C07311=1146.212,197.373,-62.411,-178.136,7.345,148.840
C07312=1146.216,197.124,-62.387,-178.138,7.343,148.841
C07313=1146.221,196.875,-62.364,-178.141,7.340,148.841
C07314=1146.225,196.626,-62.339,-178.144,7.338,148.841
C07315=1146.229,196.378,-62.315,-178.147,7.336,148.841
C07316=1146.234,196.129,-62.292,-178.149,7.334,148.842
C07317=1146.239,195.880,-62.267,-178.152,7.331,148.842
C07318=1146.244,195.631,-62.244,-178.155,7.328,148.842
C07319=1146.248,195.382,-62.220,-178.157,7.326,148.842
C07320=1146.253,195.133,-62.196,-178.161,7.324,148.843
C07321=1146.257,194.885,-62.172,-178.163,7.322,148.843
C07322=1146.261,194.635,-62.149,-178.166,7.319,148.843
C07323=1146.266,194.387,-62.124,-178.168,7.317,148.843
C07324=1146.271,194.137,-62.100,-178.172,7.314,148.844
C07325=1146.275,193.889,-62.076,-178.175,7.312,148.844
C07326=1146.280,193.640,-62.053,-178.177,7.310,148.844
C07327=1146.285,193.392,-62.029,-178.180,7.307,148.844
C07328=1146.289,193.143,-62.006,-178.183,7.305,148.845
C07329=1146.294,192.894,-61.982,-178.186,7.303,148.845
C07330=1146.298,192.645,-61.958,-178.188,7.300,148.845
C07331=1146.303,192.397,-61.934,-178.192,7.298,148.845
C07332=1146.307,192.148,-61.911,-178.194,7.296,148.845
C07333=1146.312,191.899,-61.887,-178.197,7.293,148.846
C07334=1146.317,191.650,-61.863,-178.199,7.291,148.846
C07335=1146.321,191.401,-61.840,-178.203,7.289,148.846
C07336=1146.326,191.152,-61.817,-178.205,7.287,148.846
C07337=1146.330,190.904,-61.793,-178.208,7.284,148.847
C07338=1146.335,190.655,-61.769,-178.211,7.281,148.847
C07339=1146.340,190.406,-61.746,-178.213,7.279,148.847
C07340=1146.344,190.157,-61.722,-178.216,7.276,148.847
C07341=1146.349,189.908,-61.698,-178.219,7.275,148.848
C07342=1146.354,189.659,-61.675,-178.222,7.272,148.848
C07343=1146.358,189.410,-61.652,-178.224,7.270,148.848
C07344=1146.363,189.162,-61.628,-178.228,7.267,148.848
C07345=1146.367,188.913,-61.604,-178.230,7.265,148.849
C07346=1146.372,188.664,-61.581,-178.233,7.263,148.849
C07347=1146.377,188.415,-61.558,-178.235,7.261,148.849
C07348=1146.381,188.166,-61.533,-178.239,7.258,148.849
C07349=1146.386,187.917,-61.510,-178.241,7.256,148.850
C07350=1146.391,187.668,-61.487,-178.244,7.254,148.850
C07351=1146.395,187.419,-61.463,-178.247,7.252,148.850
C07352=1146.399,187.170,-61.441,-178.250,7.249,148.850
C07353=1146.404,186.921,-61.417,-178.252,7.247,148.851
C07354=1146.409,186.672,-61.394,-178.255,7.244,148.851
C07355=1146.413,186.424,-61.370,-178.258,7.243,148.851
C07356=1146.418,186.175,-61.346,-178.261,7.240,148.851
C07357=1146.422,185.926,-61.323,-178.263,7.238,148.852
C07358=1146.426,185.677,-61.300,-178.267,7.235,148.852
C07359=1146.431,185.428,-61.277,-178.269,7.233,148.852
C07360=1146.436,185.180,-61.254,-178.272,7.231,148.853
C07361=1146.441,184.931,-61.231,-178.274,7.229,148.853
C07362=1146.446,184.682,-61.207,-178.278,7.226,148.853
C07363=1146.450,184.433,-61.184,-178.280,7.224,148.853
C07364=1146.454,184.184,-61.161,-178.283,7.221,148.853
C07365=1146.460,183.914,-61.136,-178.286,7.220,148.854
C07366=1146.465,183.644,-61.111,-178.289,7.217,148.854
C07367=1146.469,183.376,-61.086,-178.292,7.214,148.854
C07368=1146.475,183.106,-61.061,-178.295,7.212,148.855
C07369=1146.479,182.857,-61.037,-178.298,7.210,148.855
C07370=1146.484,182.608,-61.014,-178.301,7.207,148.855
C07371=1146.488,182.359,-60.991,-178.303,7.205,148.856
C07372=1146.493,182.110,-60.968,-178.307,7.203,148.856
C07373=1146.498,181.860,-60.945,-178.309,7.201,148.856
C07374=1146.502,181.612,-60.923,-178.312,7.198,148.856
C07375=1146.507,181.363,-60.900,-178.315,7.196,148.857
C07376=1146.512,181.114,-60.876,-178.317,7.194,148.857
C07377=1146.516,180.866,-60.853,-178.320,7.192,148.857
C07378=1146.520,180.617,-60.830,-178.323,7.190,148.857
C07379=1146.525,180.367,-60.807,-178.326,7.187,148.858
C07380=1146.530,180.119,-60.785,-178.329,7.185,148.858
C07381=1146.535,179.870,-60.762,-178.331,7.182,148.858
C07382=1146.539,179.621,-60.738,-178.334,7.181,148.859
C07383=1146.543,179.372,-60.716,-178.337,7.178,148.859
C07384=1146.548,179.122,-60.693,-178.340,7.176,148.859
C07385=1146.553,178.874,-60.671,-178.342,7.174,148.859
C07386=1146.558,178.625,-60.647,-178.346,7.172,148.860
C07387=1146.562,178.376,-60.624,-178.348,7.170,148.860
C07388=1146.566,178.127,-60.602,-178.351,7.167,148.860
C07389=1146.572,177.879,-60.579,-178.354,7.165,148.861
C07390=1146.576,177.630,-60.556,-178.357,7.163,148.861
C07391=1146.581,177.380,-60.533,-178.359,7.161,148.861
C07392=1146.585,177.132,-60.511,-178.362,7.159,148.861
C07393=1146.590,176.883,-60.488,-178.365,7.156,148.862
C07394=1146.594,176.634,-60.466,-178.368,7.154,148.862
C07395=1146.599,176.385,-60.442,-178.371,7.152,148.862
C07396=1146.603,176.135,-60.420,-178.373,7.150,148.862
C07397=1146.609,175.887,-60.397,-178.376,7.147,148.863
C07398=1146.613,175.638,-60.374,-178.379,7.146,148.863
C07399=1146.618,175.389,-60.352,-178.381,7.143,148.863
C07400=1146.622,175.141,-60.329,-178.385,7.141,148.864
C07401=1146.627,174.891,-60.307,-178.387,7.139,148.864
C07402=1146.631,174.642,-60.284,-178.390,7.136,148.864
C07403=1146.637,174.393,-60.262,-178.393,7.135,148.864
C07404=1146.641,174.145,-60.239,-178.395,7.133,148.865
C07405=1146.646,173.895,-60.216,-178.398,7.130,148.865
C07406=1146.650,173.647,-60.194,-178.401,7.128,148.865
C07407=1146.655,173.397,-60.171,-178.404,7.126,148.866
C07408=1146.659,173.149,-60.148,-178.406,7.124,148.866
C07409=1146.664,172.900,-60.127,-178.409,7.122,148.866
C07410=1146.669,172.651,-60.103,-178.412,7.119,148.867
C07411=1146.673,172.402,-60.081,-178.415,7.118,148.867
C07412=1146.679,172.153,-60.059,-178.418,7.115,148.867
C07413=1146.683,171.904,-60.036,-178.421,7.113,148.867
C07414=1146.687,171.655,-60.014,-178.423,7.111,148.868
C07415=1146.692,171.406,-59.991,-178.426,7.108,148.868
C07416=1146.696,171.157,-59.969,-178.429,7.107,148.868
C07417=1146.701,170.908,-59.948,-178.432,7.105,148.869
C07418=1146.706,170.659,-59.924,-178.435,7.102,148.869
C07419=1146.710,170.410,-59.902,-178.437,7.100,148.869
C07420=1146.715,170.161,-59.881,-178.440,7.098,148.870
C07421=1146.720,169.912,-59.857,-178.443,7.096,148.870
C07422=1146.725,169.664,-59.835,-178.445,7.094,148.870
C07423=1146.729,169.414,-59.813,-178.449,7.091,148.870
C07424=1146.735,169.165,-59.791,-178.451,7.090,148.871
C07425=1146.739,168.917,-59.768,-178.454,7.088,148.871
C07426=1146.743,168.667,-59.746,-178.457,7.085,148.871
C07427=1146.748,168.419,-59.725,-178.460,7.083,148.872
C07428=1146.753,168.169,-59.702,-178.462,7.081,148.872
C07429=1146.757,167.921,-59.680,-178.466,7.079,148.872
C07430=1146.761,167.672,-59.658,-178.468,7.077,148.872
C07431=1146.766,167.423,-59.636,-178.471,7.074,148.873
C07432=1146.771,167.173,-59.613,-178.474,7.073,148.873
C07433=1146.776,166.925,-59.592,-178.476,7.071,148.874
C07434=1146.781,166.675,-59.569,-178.479,7.068,148.874
C07435=1146.785,166.427,-59.548,-178.482,7.066,148.874
C07436=1146.790,166.178,-59.524,-178.485,7.065,148.874
C07437=1146.795,165.929,-59.503,-178.488,7.062,148.875
C07438=1146.799,165.680,-59.481,-178.490,7.060,148.875
C07439=1146.804,165.431,-59.459,-178.493,7.058,148.875
C07440=1146.808,165.182,-59.437,-178.496,7.056,148.876
C07441=1146.813,164.933,-59.415,-178.499,7.054,148.876
C07442=1146.817,164.684,-59.393,-178.501,7.052,148.876
C07443=1146.823,164.435,-59.371,-178.504,7.049,148.877
C07444=1146.827,164.185,-59.349,-178.507,7.048,148.877
C07445=1146.832,163.937,-59.327,-178.510,7.046,148.877
C07446=1146.837,163.687,-59.305,-178.513,7.043,148.878
C07447=1146.841,163.439,-59.284,-178.515,7.041,148.878
C07448=1146.846,163.189,-59.261,-178.518,7.039,148.878
C07449=1146.851,162.941,-59.240,-178.521,7.038,148.879
C07450=1146.855,162.692,-59.218,-178.524,7.035,148.879
C07451=1146.860,162.443,-59.196,-178.526,7.033,148.879
C07452=1146.865,162.194,-59.174,-178.529,7.031,148.879
C07453=1146.869,161.945,-59.152,-178.532,7.029,148.880
C07454=1146.874,161.696,-59.131,-178.535,7.027,148.880
C07455=1146.879,161.447,-59.108,-178.538,7.025,148.881
C07456=1146.884,161.198,-59.086,-178.540,7.023,148.881
C07457=1146.889,160.949,-59.065,-178.543,7.021,148.881
C07458=1146.893,160.699,-59.043,-178.546,7.019,148.881
C07459=1146.898,160.451,-59.022,-178.549,7.017,148.882
C07460=1146.902,160.201,-59.000,-178.552,7.015,148.882
C07461=1146.907,159.953,-58.978,-178.554,7.013,148.882
C07462=1146.912,159.704,-58.956,-178.557,7.011,148.883
C07463=1146.916,159.454,-58.935,-178.560,7.008,148.883
C07464=1146.921,159.206,-58.914,-178.563,7.007,148.883
C07465=1146.925,158.957,-58.892,-178.565,7.005,148.884
C07466=1146.930,158.708,-58.870,-178.569,7.003,148.884
C07467=1146.935,158.459,-58.848,-178.571,7.000,148.884
C07468=1146.939,158.209,-58.827,-178.574,6.999,148.885
C07469=1146.944,157.940,-58.803,-178.577,6.996,148.885
C07470=1146.950,157.672,-58.781,-178.580,6.994,148.886
C07471=1146.955,157.403,-58.757,-178.583,6.992,148.886
C07472=1146.960,157.134,-58.734,-178.586,6.990,148.886
C07473=1146.964,156.884,-58.712,-178.588,6.988,148.887
C07474=1146.969,156.636,-58.691,-178.592,6.986,148.887
C07475=1146.974,156.387,-58.669,-178.594,6.984,148.887
C07476=1146.978,156.137,-58.648,-178.597,6.982,148.888
C07477=1146.983,155.889,-58.626,-178.600,6.980,148.888
C07478=1146.989,155.639,-58.605,-178.603,6.978,148.888
C07479=1146.993,155.391,-58.584,-178.605,6.976,148.889
C07480=1146.997,155.142,-58.562,-178.608,6.974,148.889
C07481=1147.002,154.892,-58.541,-178.611,6.972,148.889
C07482=1147.007,154.644,-58.519,-178.614,6.970,148.890
C07483=1147.012,154.394,-58.498,-178.616,6.968,148.890
C07484=1147.016,154.145,-58.476,-178.619,6.966,148.890
C07485=1147.021,153.896,-58.456,-178.622,6.964,148.891
C07486=1147.026,153.647,-58.434,-178.625,6.962,148.891
C07487=1147.030,153.398,-58.413,-178.628,6.960,148.891
C07488=1147.035,153.149,-58.391,-178.630,6.959,148.892
C07489=1147.040,152.900,-58.371,-178.633,6.957,148.892
C07490=1147.044,152.651,-58.349,-178.636,6.954,148.892
C07491=1147.050,152.402,-58.328,-178.639,6.952,148.893
C07492=1147.054,152.153,-58.306,-178.641,6.951,148.893
C07493=1147.058,151.904,-58.286,-178.644,6.949,148.893
C07494=1147.063,151.655,-58.264,-178.647,6.946,148.894
C07495=1147.068,151.406,-58.243,-178.650,6.945,148.894
C07496=1147.073,151.157,-58.221,-178.653,6.943,148.895
C07497=1147.077,150.908,-58.201,-178.655,6.941,148.895
C07498=1147.082,150.658,-58.180,-178.658,6.938,148.895
C07499=1147.087,150.410,-58.158,-178.661,6.937,148.896
C07500=1147.092,150.161,-58.138,-178.664,6.935,148.896
C07501=1147.097,149.911,-58.117,-178.666,6.933,148.896
C07502=1147.101,149.662,-58.095,-178.669,6.931,148.897
C07503=1147.105,149.413,-58.074,-178.672,6.929,148.897
C07504=1147.111,149.164,-58.053,-178.675,6.927,148.897
C07505=1147.115,148.915,-58.032,-178.677,6.925,148.898
C07506=1147.120,148.666,-58.011,-178.680,6.923,148.898
C07507=1147.125,148.417,-57.990,-178.683,6.922,148.898
C07508=1147.129,148.168,-57.968,-178.686,6.919,148.899
C07509=1147.134,147.919,-57.948,-178.689,6.917,148.899
C07510=1147.139,147.670,-57.927,-178.691,6.916,148.899
C07511=1147.143,147.421,-57.907,-178.694,6.914,148.900
C07512=1147.149,147.171,-57.886,-178.697,6.912,148.900
C07513=1147.153,146.923,-57.864,-178.700,6.910,148.901
C07514=1147.158,146.674,-57.844,-178.703,6.908,148.901
C07515=1147.163,146.424,-57.823,-178.705,6.906,148.901
C07516=1147.168,146.176,-57.802,-178.708,6.904,148.902
C07517=1147.172,145.926,-57.781,-178.711,6.903,148.902
C07518=1147.176,145.677,-57.760,-178.713,6.901,148.902
C07519=1147.181,145.428,-57.739,-178.717,6.898,148.903
C07520=1147.186,145.179,-57.718,-178.719,6.897,148.903
C07521=1147.191,144.930,-57.697,-178.722,6.895,148.903
C07522=1147.195,144.681,-57.677,-178.725,6.893,148.904
C07523=1147.201,144.432,-57.656,-178.727,6.891,148.904
C07524=1147.205,144.183,-57.636,-178.731,6.889,148.905
C07525=1147.210,143.933,-57.615,-178.733,6.887,148.905
C07526=1147.215,143.684,-57.594,-178.736,6.886,148.905
C07527=1147.220,143.435,-57.573,-178.739,6.884,148.906
C07528=1147.224,143.186,-57.553,-178.741,6.882,148.906
C07529=1147.229,142.938,-57.531,-178.744,6.880,148.906
C07530=1147.234,142.689,-57.511,-178.747,6.878,148.907
C07531=1147.239,142.439,-57.490,-178.750,6.876,148.907
C07532=1147.243,142.190,-57.470,-178.753,6.874,148.907
C07533=1147.248,141.941,-57.449,-178.755,6.872,148.908
C07534=1147.252,141.691,-57.428,-178.758,6.871,148.908
C07535=1147.257,141.442,-57.408,-178.761,6.869,148.909
C07536=1147.262,141.193,-57.387,-178.763,6.867,148.909
C07537=1147.267,140.944,-57.367,-178.767,6.865,148.909
C07538=1147.271,140.695,-57.347,-178.769,6.863,148.910
C07539=1147.276,140.445,-57.326,-178.772,6.861,148.910
C07540=1147.281,140.197,-57.305,-178.775,6.860,148.911
C07541=1147.286,139.948,-57.285,-178.778,6.858,148.911
C07542=1147.291,139.699,-57.264,-178.780,6.856,148.911
C07543=1147.295,139.450,-57.244,-178.783,6.854,148.912
C07544=1147.300,139.201,-57.223,-178.786,6.852,148.912
C07545=1147.305,138.951,-57.203,-178.789,6.850,148.913
C07546=1147.310,138.702,-57.183,-178.792,6.848,148.913
C07547=1147.314,138.453,-57.163,-178.794,6.847,148.913
C07548=1147.319,138.204,-57.142,-178.797,6.845,148.914
C07549=1147.324,137.955,-57.121,-178.799,6.843,148.914
C07550=1147.328,137.706,-57.102,-178.802,6.841,148.914
C07551=1147.334,137.456,-57.081,-178.805,6.840,148.915
C07552=1147.338,137.207,-57.060,-178.807,6.838,148.915
C07553=1147.342,136.958,-57.040,-178.811,6.835,148.915
C07554=1147.347,136.709,-57.019,-178.814,6.834,148.916
C07555=1147.352,136.460,-56.999,-178.816,6.832,148.916
C07556=1147.357,136.211,-56.979,-178.819,6.830,148.917
C07557=1147.362,135.962,-56.959,-178.822,6.829,148.917
C07558=1147.367,135.713,-56.939,-178.824,6.827,148.917
C07559=1147.372,135.464,-56.918,-178.827,6.825,148.918
C07560=1147.376,135.215,-56.898,-178.830,6.823,148.918
C07561=1147.381,134.965,-56.878,-178.833,6.822,148.919
C07562=1147.385,134.716,-56.858,-178.836,6.819,148.919
C07563=1147.390,134.467,-56.837,-178.839,6.817,148.919
C07564=1147.395,134.217,-56.817,-178.841,6.816,148.920
C07565=1147.400,133.969,-56.797,-178.844,6.814,148.920
C07566=1147.405,133.720,-56.777,-178.847,6.812,148.920
C07567=1147.410,133.471,-56.757,-178.849,6.811,148.921
C07568=1147.414,133.222,-56.737,-178.852,6.809,148.921
C07569=1147.419,132.972,-56.717,-178.855,6.807,148.922
C07570=1147.424,132.723,-56.696,-178.858,6.805,148.922
C07571=1147.429,132.473,-56.676,-178.860,6.804,148.922
C07572=1147.434,132.225,-56.656,-178.863,6.802,148.923
C07573=1147.439,131.956,-56.635,-178.866,6.800,148.923
C07574=1147.444,131.688,-56.613,-178.869,6.798,148.924
C07575=1147.449,131.419,-56.592,-178.872,6.797,148.924
C07576=1147.454,131.150,-56.570,-178.875,6.794,148.925
C07577=1147.459,130.901,-56.550,-178.878,6.792,148.925
C07578=1147.464,130.652,-56.530,-178.881,6.791,148.925
C07579=1147.468,130.403,-56.510,-178.884,6.789,148.926
C07580=1147.473,130.154,-56.491,-178.886,6.787,148.926
C07581=1147.478,129.905,-56.470,-178.889,6.785,148.927
C07582=1147.483,129.655,-56.451,-178.892,6.784,148.927
C07583=1147.487,129.406,-56.431,-178.895,6.782,148.927
C07584=1147.492,129.158,-56.411,-178.897,6.780,148.928
C07585=1147.497,128.908,-56.391,-178.900,6.779,148.928
C07586=1147.502,128.659,-56.371,-178.903,6.777,148.929
C07587=1147.506,128.410,-56.351,-178.905,6.775,148.929
C07588=1147.512,128.161,-56.332,-178.908,6.774,148.929
C07589=1147.516,127.912,-56.312,-178.911,6.772,148.930
C07590=1147.521,127.662,-56.292,-178.914,6.770,148.930
C07591=1147.526,127.413,-56.272,-178.916,6.768,148.931
C07592=1147.531,127.164,-56.252,-178.919,6.767,148.931
C07593=1147.535,126.915,-56.233,-178.922,6.764,148.931
C07594=1147.540,126.665,-56.213,-178.925,6.762,148.932
C07595=1147.545,126.416,-56.193,-178.928,6.761,148.932
C07596=1147.550,126.167,-56.173,-178.931,6.759,148.933
C07597=1147.555,125.918,-56.154,-178.934,6.758,148.933
C07598=1147.559,125.668,-56.134,-178.936,6.756,148.934
C07599=1147.565,125.419,-56.115,-178.939,6.754,148.934
C07600=1147.568,125.171,-56.095,-178.942,6.753,148.934
C07601=1147.573,124.921,-56.075,-178.945,6.751,148.935
C07602=1147.579,124.672,-56.056,-178.947,6.749,148.935
C07603=1147.583,124.423,-56.036,-178.950,6.748,148.936
C07604=1147.588,124.173,-56.017,-178.953,6.746,148.936
C07605=1147.593,123.925,-55.997,-178.955,6.744,148.936
C07606=1147.598,123.675,-55.977,-178.958,6.742,148.937
C07607=1147.603,123.426,-55.957,-178.961,6.741,148.937
C07608=1147.607,123.177,-55.939,-178.964,6.739,148.938
C07609=1147.612,122.928,-55.919,-178.966,6.737,148.938
C07610=1147.617,122.678,-55.899,-178.969,6.736,148.938
C07611=1147.622,122.429,-55.880,-178.972,6.734,148.939
C07612=1147.627,122.180,-55.860,-178.975,6.733,148.939
C07613=1147.630,121.931,-55.841,-178.978,6.731,148.940
C07614=1147.636,121.682,-55.821,-178.980,6.729,148.940
C07615=1147.640,121.433,-55.802,-178.983,6.727,148.941
C07616=1147.646,121.184,-55.782,-178.986,6.726,148.941
C07617=1147.651,120.934,-55.763,-178.989,6.724,148.941
C07618=1147.655,120.685,-55.744,-178.991,6.722,148.942
C07619=1147.660,120.436,-55.724,-178.994,6.721,148.942
C07620=1147.665,120.186,-55.705,-178.997,6.719,148.943
C07621=1147.670,119.938,-55.685,-178.999,6.717,148.943
C07622=1147.674,119.688,-55.666,-179.002,6.716,148.943
C07623=1147.679,119.439,-55.647,-179.005,6.714,148.944
C07624=1147.684,119.190,-55.627,-179.008,6.713,148.944
C07625=1147.689,118.940,-55.608,-179.011,6.711,148.945
C07626=1147.693,118.692,-55.589,-179.014,6.709,148.945
C07627=1147.699,118.442,-55.570,-179.016,6.707,148.946
C07628=1147.704,118.193,-55.551,-179.019,6.706,148.946
C07629=1147.708,117.943,-55.532,-179.022,6.704,148.946
C07630=1147.713,117.695,-55.512,-179.024,6.702,148.947
C07631=1147.718,117.445,-55.493,-179.027,6.701,148.947
C07632=1147.723,117.196,-55.474,-179.029,6.700,148.948
C07633=1147.727,116.947,-55.454,-179.032,6.698,148.948
C07634=1147.733,116.698,-55.435,-179.035,6.696,148.948
C07635=1147.737,116.448,-55.417,-179.038,6.695,148.949
C07636=1147.742,116.199,-55.397,-179.041,6.693,148.950
C07637=1147.747,115.950,-55.378,-179.043,6.692,148.950
C07638=1147.751,115.700,-55.359,-179.046,6.690,148.950
C07639=1147.756,115.452,-55.339,-179.049,6.688,148.951
C07640=1147.761,115.202,-55.321,-179.052,6.687,148.951
C07641=1147.766,114.953,-55.302,-179.054,6.685,148.952
C07642=1147.771,114.704,-55.283,-179.057,6.683,148.952
C07643=1147.775,114.455,-55.263,-179.060,6.681,148.952
C07644=1147.781,114.205,-55.245,-179.063,6.680,148.953
C07645=1147.785,113.956,-55.226,-179.066,6.678,148.953
C07646=1147.790,113.707,-55.207,-179.068,6.677,148.954
C07647=1147.795,113.458,-55.187,-179.071,6.675,148.954
C07648=1147.800,113.208,-55.169,-179.074,6.673,148.955
C07649=1147.805,112.959,-55.149,-179.077,6.672,148.955
C07650=1147.809,112.710,-55.131,-179.079,6.671,148.955
C07651=1147.814,112.460,-55.112,-179.081,6.669,148.956
C07652=1147.819,112.212,-55.093,-179.085,6.668,148.956
C07653=1147.824,111.963,-55.074,-179.087,6.666,148.957
C07654=1147.829,111.713,-55.055,-179.090,6.664,148.957
C07655=1147.834,111.464,-55.036,-179.093,6.663,148.958
C07656=1147.838,111.214,-55.018,-179.095,6.661,148.958
C07657=1147.844,110.965,-54.998,-179.098,6.659,148.958
C07658=1147.848,110.717,-54.980,-179.101,6.658,148.959
C07659=1147.853,110.466,-54.961,-179.104,6.656,148.960
C07660=1147.858,110.218,-54.942,-179.107,6.655,148.960
C07661=1147.863,109.968,-54.923,-179.110,6.653,148.960
C07662=1147.868,109.719,-54.904,-179.112,6.652,148.961
C07663=1147.873,109.470,-54.886,-179.114,6.650,148.961
C07664=1147.877,109.220,-54.867,-179.117,6.649,148.962
C07665=1147.882,108.971,-54.849,-179.120,6.647,148.962
C07666=1147.888,108.722,-54.829,-179.123,6.646,148.963
C07667=1147.892,108.472,-54.811,-179.126,6.644,148.963
C07668=1147.896,108.224,-54.792,-179.129,6.642,148.963
C07669=1147.901,107.974,-54.773,-179.131,6.641,148.964
C07670=1147.906,107.725,-54.755,-179.134,6.639,148.964
C07671=1147.912,107.476,-54.736,-179.137,6.637,148.965
C07672=1147.916,107.226,-54.717,-179.139,6.637,148.965
C07673=1147.921,106.977,-54.699,-179.142,6.635,148.966
C07674=1147.926,106.728,-54.680,-179.145,6.633,148.966
C07675=1147.930,106.478,-54.662,-179.148,6.632,148.967
C07676=1147.935,106.229,-54.644,-179.150,6.630,148.967
C07677=1147.941,105.961,-54.623,-179.153,6.629,148.968
C07678=1147.946,105.693,-54.603,-179.156,6.627,148.968
C07679=1147.951,105.424,-54.583,-179.159,6.625,148.968
C07680=1147.956,105.156,-54.564,-179.162,6.624,148.969
C07681=1147.961,104.907,-54.544,-179.165,6.622,148.969
C07682=1147.966,104.658,-54.526,-179.168,6.620,148.970
C07683=1147.971,104.408,-54.508,-179.170,6.619,148.970
C07684=1147.975,104.159,-54.489,-179.173,6.617,148.971
C07685=1147.981,103.910,-54.471,-179.176,6.615,148.971
C07686=1147.986,103.660,-54.453,-179.179,6.614,148.972
C07687=1147.990,103.411,-54.434,-179.181,6.613,148.972
C07688=1147.996,103.162,-54.415,-179.184,6.612,148.973
C07689=1148.000,102.913,-54.397,-179.187,6.610,148.973
C07690=1148.005,102.663,-54.379,-179.189,6.608,148.973
C07691=1148.010,102.413,-54.361,-179.192,6.606,148.974
C07692=1148.014,102.165,-54.342,-179.195,6.605,148.974
C07693=1148.020,101.915,-54.324,-179.198,6.603,148.975
C07694=1148.025,101.666,-54.306,-179.200,6.603,148.975
C07695=1148.029,101.416,-54.287,-179.203,6.601,148.976
C07696=1148.034,101.167,-54.269,-179.206,6.599,148.976
C07697=1148.039,100.919,-54.251,-179.209,6.598,148.977
C07698=1148.044,100.669,-54.232,-179.212,6.596,148.977
C07699=1148.049,100.420,-54.214,-179.214,6.594,148.978
C07700=1148.054,100.170,-54.196,-179.216,6.594,148.978
C07701=1148.058,99.921,-54.178,-179.219,6.592,148.978
C07702=1148.063,99.672,-54.160,-179.222,6.591,148.979
C07703=1148.068,99.423,-54.142,-179.225,6.589,148.979
C07704=1148.073,99.173,-54.124,-179.228,6.587,148.980
C07705=1148.078,98.924,-54.104,-179.231,6.586,148.980
C07706=1148.083,98.675,-54.086,-179.233,6.585,148.981
C07707=1148.088,98.426,-54.068,-179.236,6.583,148.981
C07708=1148.093,98.176,-54.050,-179.239,6.582,148.982
C07709=1148.098,97.927,-54.032,-179.241,6.580,148.982
C07710=1148.102,97.678,-54.014,-179.244,6.578,148.983
C07711=1148.107,97.428,-53.996,-179.246,6.577,148.983
C07712=1148.112,97.179,-53.978,-179.249,6.576,148.984
C07713=1148.117,96.930,-53.960,-179.252,6.574,148.984
C07714=1148.122,96.681,-53.942,-179.255,6.573,148.984
C07715=1148.126,96.431,-53.924,-179.258,6.571,148.985
C07716=1148.132,96.182,-53.905,-179.260,6.569,148.985
C07717=1148.137,95.933,-53.887,-179.263,6.569,148.986
C07718=1148.141,95.683,-53.869,-179.266,6.567,148.986
C07719=1148.146,95.434,-53.851,-179.268,6.566,148.987
C07720=1148.151,95.184,-53.834,-179.271,6.564,148.987
C07721=1148.156,94.935,-53.816,-179.274,6.563,148.988
C07722=1148.161,94.686,-53.798,-179.277,6.562,148.988
C07723=1148.166,94.436,-53.780,-179.279,6.560,148.989
C07724=1148.171,94.187,-53.762,-179.282,6.558,148.989
C07725=1148.176,93.938,-53.744,-179.285,6.557,148.990
C07726=1148.181,93.689,-53.726,-179.288,6.555,148.990
C07727=1148.186,93.440,-53.708,-179.290,6.554,148.991
C07728=1148.191,93.190,-53.691,-179.293,6.553,148.991
C07729=1148.195,92.940,-53.673,-179.296,6.551,148.991
C07730=1148.200,92.691,-53.655,-179.299,6.550,148.992
C07731=1148.204,92.442,-53.637,-179.301,6.549,148.992
C07732=1148.209,92.193,-53.619,-179.304,6.547,148.993
C07733=1148.215,91.943,-53.602,-179.306,6.545,148.993
C07734=1148.219,91.694,-53.584,-179.310,6.544,148.994
C07735=1148.224,91.445,-53.566,-179.312,6.542,148.994
C07736=1148.229,91.195,-53.548,-179.314,6.542,148.995
C07737=1148.234,90.946,-53.530,-179.317,6.540,148.995
C07738=1148.239,90.696,-53.513,-179.320,6.539,148.996
C07739=1148.244,90.447,-53.495,-179.323,6.537,148.996
C07740=1148.249,90.198,-53.477,-179.325,6.536,148.997
C07741=1148.254,89.949,-53.460,-179.328,6.534,148.997
C07742=1148.259,89.699,-53.442,-179.331,6.533,148.998
C07743=1148.264,89.450,-53.424,-179.334,6.531,148.998
C07744=1148.269,89.200,-53.407,-179.336,6.531,148.999
C07745=1148.274,88.951,-53.389,-179.339,6.529,148.999
C07746=1148.279,88.702,-53.371,-179.342,6.527,148.999
C07747=1148.283,88.453,-53.354,-179.345,6.526,149.000
C07748=1148.288,88.203,-53.336,-179.347,6.525,149.001
C07749=1148.293,87.954,-53.318,-179.350,6.523,149.001
C07750=1148.298,87.705,-53.301,-179.352,6.522,149.001
C07751=1148.303,87.455,-53.283,-179.356,6.520,149.002
C07752=1148.308,87.206,-53.266,-179.358,6.519,149.002
C07753=1148.312,86.957,-53.248,-179.361,6.518,149.003
C07754=1148.317,86.707,-53.230,-179.364,6.516,149.004
C07755=1148.323,86.458,-53.213,-179.367,6.515,149.004
C07756=1148.327,86.209,-53.196,-179.369,6.514,149.004
C07757=1148.333,85.960,-53.179,-179.371,6.512,149.005
C07758=1148.337,85.711,-53.161,-179.375,6.511,149.005
C07759=1148.343,85.461,-53.143,-179.377,6.510,149.006
C07760=1148.347,85.212,-53.126,-179.379,6.508,149.006
C07761=1148.352,84.962,-53.109,-179.382,6.507,149.007
C07762=1148.357,84.713,-53.091,-179.385,6.505,149.007
C07763=1148.362,84.463,-53.074,-179.388,6.505,149.008
C07764=1148.366,84.214,-53.056,-179.390,6.503,149.008
C07765=1148.372,83.964,-53.039,-179.393,6.501,149.009
C07766=1148.377,83.715,-53.021,-179.396,6.500,149.009
C07767=1148.381,83.466,-53.004,-179.398,6.499,149.010
C07768=1148.387,83.217,-52.987,-179.401,6.497,149.010
C07769=1148.392,82.968,-52.969,-179.404,6.496,149.011
C07770=1148.396,82.718,-52.953,-179.407,6.495,149.011
C07771=1148.401,82.469,-52.935,-179.409,6.494,149.012
C07772=1148.406,82.219,-52.917,-179.412,6.492,149.012
C07773=1148.411,81.970,-52.901,-179.415,6.491,149.013
C07774=1148.416,81.720,-52.883,-179.417,6.490,149.013
C07775=1148.420,81.471,-52.866,-179.420,6.488,149.014
C07776=1148.426,81.222,-52.849,-179.423,6.487,149.014
C07777=1148.431,80.973,-52.831,-179.425,6.486,149.015
C07778=1148.435,80.723,-52.815,-179.428,6.484,149.015
C07779=1148.441,80.473,-52.797,-179.431,6.482,149.016
C07780=1148.446,80.224,-52.779,-179.434,6.482,149.016
C07781=1148.451,79.956,-52.762,-179.436,6.480,149.017
C07782=1148.456,79.687,-52.743,-179.440,6.479,149.017
C07783=1148.461,79.419,-52.725,-179.442,6.477,149.018
C07784=1148.467,79.151,-52.706,-179.446,6.476,149.018
C07785=1148.472,78.902,-52.689,-179.448,6.474,149.019
C07786=1148.476,78.652,-52.672,-179.450,6.473,149.019
C07787=1148.481,78.402,-52.655,-179.453,6.472,149.020
C07788=1148.487,78.154,-52.638,-179.456,6.471,149.020
C07789=1148.492,77.904,-52.621,-179.459,6.470,149.021
C07790=1148.496,77.655,-52.604,-179.461,6.468,149.021
C07791=1148.501,77.405,-52.586,-179.464,6.467,149.022
C07792=1148.506,77.156,-52.570,-179.467,6.466,149.022
C07793=1148.511,76.906,-52.553,-179.469,6.464,149.023
C07794=1148.516,76.657,-52.536,-179.472,6.462,149.023
C07795=1148.521,76.407,-52.519,-179.475,6.462,149.024
C07796=1148.525,76.158,-52.501,-179.477,6.460,149.024
C07797=1148.531,75.909,-52.485,-179.480,6.459,149.025
C07798=1148.536,75.660,-52.468,-179.483,6.458,149.025
C07799=1148.541,75.410,-52.451,-179.486,6.456,149.026
C07800=1148.545,75.160,-52.434,-179.488,6.455,149.026
C07801=1148.551,74.911,-52.417,-179.491,6.454,149.027
C07802=1148.556,74.662,-52.400,-179.494,6.453,149.027
C07803=1148.560,74.412,-52.384,-179.496,6.451,149.028
C07804=1148.566,74.163,-52.367,-179.499,6.450,149.028
C07805=1148.570,73.914,-52.350,-179.502,6.449,149.029
C07806=1148.576,73.664,-52.333,-179.504,6.448,149.029
C07807=1148.580,73.415,-52.316,-179.507,6.447,149.030
C07808=1148.585,73.166,-52.300,-179.510,6.445,149.030
C07809=1148.590,72.916,-52.283,-179.512,6.444,149.031
C07810=1148.595,72.667,-52.266,-179.515,6.442,149.031
C07811=1148.601,72.417,-52.249,-179.518,6.441,149.032
C07812=1148.605,72.168,-52.232,-179.520,6.440,149.032
C07813=1148.610,71.918,-52.216,-179.523,6.439,149.033
C07814=1148.615,71.669,-52.199,-179.526,6.437,149.033
C07815=1148.620,71.420,-52.182,-179.528,6.436,149.034
C07816=1148.624,71.170,-52.166,-179.531,6.435,149.034
C07817=1148.630,70.921,-52.149,-179.534,6.434,149.035
C07818=1148.635,70.672,-52.132,-179.536,6.433,149.035
C07819=1148.639,70.422,-52.115,-179.539,6.431,149.036
C07820=1148.645,70.173,-52.098,-179.542,6.431,149.036
C07821=1148.649,69.924,-52.082,-179.545,6.429,149.037
C07822=1148.654,69.674,-52.065,-179.547,6.427,149.037
C07823=1148.659,69.425,-52.049,-179.550,6.427,149.038
C07824=1148.665,69.175,-52.032,-179.553,6.425,149.038
C07825=1148.670,68.926,-52.016,-179.555,6.424,149.039
C07826=1148.674,68.677,-51.999,-179.558,6.423,149.039
C07827=1148.679,68.427,-51.982,-179.561,6.421,149.040
C07828=1148.684,68.178,-51.966,-179.563,6.420,149.040
C07829=1148.689,67.928,-51.950,-179.566,6.419,149.041
C07830=1148.694,67.679,-51.933,-179.568,6.418,149.041
C07831=1148.699,67.430,-51.917,-179.571,6.417,149.042
C07832=1148.704,67.180,-51.899,-179.574,6.415,149.042
C07833=1148.709,66.931,-51.883,-179.576,6.414,149.043
C07834=1148.714,66.681,-51.867,-179.579,6.413,149.043
C07835=1148.719,66.432,-51.851,-179.582,6.412,149.044
C07836=1148.723,66.183,-51.834,-179.585,6.411,149.044
C07837=1148.729,65.933,-51.817,-179.587,6.409,149.045
C07838=1148.734,65.684,-51.801,-179.590,6.408,149.045
C07839=1148.739,65.434,-51.785,-179.593,6.407,149.046
C07840=1148.744,65.185,-51.768,-179.595,6.406,149.046
C07841=1148.748,64.935,-51.752,-179.598,6.405,149.047
C07842=1148.754,64.686,-51.736,-179.600,6.404,149.047
C07843=1148.759,64.437,-51.719,-179.603,6.402,149.048
C07844=1148.764,64.187,-51.703,-179.606,6.401,149.049
C07845=1148.769,63.938,-51.687,-179.608,6.400,149.049
C07846=1148.773,63.688,-51.670,-179.611,6.398,149.049
C07847=1148.778,63.439,-51.654,-179.614,6.398,149.050
C07848=1148.783,63.189,-51.638,-179.616,6.396,149.050
C07849=1148.788,62.940,-51.622,-179.619,6.396,149.051
C07850=1148.793,62.691,-51.605,-179.622,6.394,149.052
C07851=1148.799,62.442,-51.589,-179.625,6.392,149.052
C07852=1148.803,62.191,-51.573,-179.627,6.392,149.053
C07853=1148.808,61.943,-51.556,-179.630,6.390,149.053
C07854=1148.813,61.693,-51.540,-179.632,6.389,149.054
C07855=1148.818,61.444,-51.524,-179.635,6.388,149.054
C07856=1148.823,61.194,-51.508,-179.638,6.387,149.055
C07857=1148.828,60.945,-51.492,-179.640,6.386,149.055
C07858=1148.834,60.695,-51.476,-179.643,6.385,149.056
C07859=1148.838,60.446,-51.460,-179.646,6.383,149.056
C07860=1148.843,60.197,-51.444,-179.648,6.382,149.057
C07861=1148.848,59.947,-51.427,-179.651,6.381,149.057
C07862=1148.853,59.698,-51.412,-179.654,6.380,149.058
C07863=1148.858,59.448,-51.395,-179.656,6.379,149.058
C07864=1148.863,59.199,-51.379,-179.659,6.377,149.059
C07865=1148.868,58.949,-51.363,-179.661,6.377,149.059
C07866=1148.873,58.700,-51.347,-179.665,6.375,149.060
C07867=1148.878,58.450,-51.330,-179.667,6.374,149.060
C07868=1148.883,58.201,-51.315,-179.669,6.373,149.061
C07869=1148.888,57.952,-51.299,-179.672,6.372,149.061
C07870=1148.893,57.702,-51.283,-179.675,6.371,149.062
C07871=1148.898,57.453,-51.267,-179.677,6.370,149.062
C07872=1148.903,57.203,-51.250,-179.680,6.369,149.063
C07873=1148.908,56.954,-51.235,-179.683,6.367,149.063
C07874=1148.913,56.704,-51.219,-179.686,6.366,149.064
C07875=1148.918,56.455,-51.203,-179.688,6.365,149.065
C07876=1148.923,56.206,-51.187,-179.691,6.364,149.065
C07877=1148.928,55.955,-51.171,-179.694,6.363,149.066
C07878=1148.933,55.707,-51.155,-179.696,6.362,149.066
C07879=1148.939,55.457,-51.139,-179.699,6.360,149.067
C07880=1148.943,55.207,-51.124,-179.701,6.360,149.067
C07881=1148.948,54.959,-51.107,-179.704,6.358,149.068
C07882=1148.953,54.709,-51.092,-179.707,6.358,149.068
C07883=1148.958,54.459,-51.076,-179.709,6.356,149.069
C07884=1148.963,54.210,-51.060,-179.712,6.355,149.069
C07885=1148.968,53.942,-51.043,-179.715,6.354,149.070
C07886=1148.974,53.672,-51.026,-179.718,6.352,149.070
C07887=1148.979,53.404,-51.009,-179.720,6.352,149.071
C07888=1148.985,53.135,-50.992,-179.723,6.350,149.072
C07889=1148.990,52.886,-50.976,-179.726,6.349,149.072
C07890=1148.994,52.637,-50.960,-179.728,6.348,149.073
C07891=1148.999,52.387,-50.945,-179.731,6.347,149.073
C07892=1149.005,52.138,-50.929,-179.734,6.346,149.074
C07893=1149.010,51.888,-50.913,-179.736,6.345,149.074
C07894=1149.015,51.639,-50.897,-179.739,6.344,149.075
C07895=1149.019,51.390,-50.882,-179.741,6.343,149.075
C07896=1149.025,51.140,-50.866,-179.745,6.341,149.076
C07897=1149.029,50.890,-50.850,-179.747,6.341,149.076
C07898=1149.035,50.641,-50.835,-179.749,6.339,149.077
C07899=1149.039,50.392,-50.820,-179.752,6.338,149.077
C07900=1149.044,50.142,-50.804,-179.755,6.337,149.078
C07901=1149.050,49.892,-50.788,-179.757,6.336,149.079
C07902=1149.055,49.644,-50.772,-179.760,6.335,149.079
C07903=1149.059,49.394,-50.757,-179.762,6.334,149.079
C07904=1149.064,49.144,-50.741,-179.766,6.333,149.080
C07905=1149.070,48.895,-50.725,-179.768,6.332,149.081
C07906=1149.075,48.646,-50.710,-179.771,6.330,149.081
C07907=1149.079,48.396,-50.694,-179.773,6.330,149.082
C07908=1149.084,48.146,-50.679,-179.776,6.328,149.082
C07909=1149.090,47.897,-50.663,-179.779,6.327,149.083
C07910=1149.094,47.648,-50.648,-179.781,6.327,149.083
C07911=1149.099,47.398,-50.632,-179.784,6.325,149.084
C07912=1149.105,47.148,-50.617,-179.786,6.325,149.084
C07913=1149.110,46.899,-50.601,-179.789,6.323,149.085
C07914=1149.115,46.650,-50.586,-179.792,6.322,149.085
C07915=1149.120,46.400,-50.570,-179.794,6.321,149.086
C07916=1149.124,46.151,-50.555,-179.797,6.320,149.087
C07917=1149.129,45.901,-50.540,-179.800,6.319,149.087
C07918=1149.135,45.652,-50.524,-179.802,6.318,149.087
C07919=1149.139,45.403,-50.509,-179.805,6.317,149.088
C07920=1149.145,45.153,-50.493,-179.807,6.316,149.089
C07921=1149.150,44.903,-50.478,-179.810,6.315,149.089
C07922=1149.155,44.654,-50.463,-179.813,6.314,149.090
C07923=1149.160,44.404,-50.448,-179.815,6.313,149.090
C07924=1149.165,44.155,-50.432,-179.818,6.311,149.091
C07925=1149.170,43.906,-50.417,-179.820,6.311,149.091
C07926=1149.175,43.656,-50.401,-179.823,6.309,149.092
C07927=1149.179,43.406,-50.386,-179.826,6.308,149.092
C07928=1149.185,43.157,-50.370,-179.828,6.308,149.093
C07929=1149.190,42.907,-50.356,-179.831,6.306,149.093
C07930=1149.195,42.658,-50.341,-179.833,6.306,149.094
C07931=1149.201,42.409,-50.325,-179.836,6.304,149.095
C07932=1149.205,42.159,-50.310,-179.839,6.303,149.095
C07933=1149.210,41.909,-50.294,-179.841,6.302,149.095
C07934=1149.215,41.660,-50.280,-179.844,6.301,149.096
C07935=1149.220,41.410,-50.264,-179.846,6.300,149.097
C07936=1149.225,41.161,-50.249,-179.849,6.299,149.097
C07937=1149.230,40.912,-50.234,-179.851,6.298,149.098
C07938=1149.235,40.663,-50.219,-179.855,6.297,149.098
C07939=1149.241,40.413,-50.204,-179.857,6.296,149.099
C07940=1149.245,40.164,-50.189,-179.859,6.295,149.099
C07941=1149.250,39.913,-50.173,-179.862,6.294,149.100
C07942=1149.255,39.664,-50.158,-179.864,6.293,149.100
C07943=1149.260,39.414,-50.143,-179.868,6.292,149.101
C07944=1149.265,39.165,-50.128,-179.870,6.291,149.102
C07945=1149.271,38.916,-50.112,-179.873,6.290,149.102
C07946=1149.275,38.666,-50.098,-179.875,6.289,149.103
C07947=1149.281,38.417,-50.082,-179.877,6.288,149.103
C07948=1149.286,38.168,-50.067,-179.881,6.287,149.104
C07949=1149.291,37.918,-50.053,-179.883,6.286,149.104
C07950=1149.296,37.668,-50.038,-179.885,6.286,149.105
C07951=1149.301,37.419,-50.023,-179.888,6.284,149.105
C07952=1149.306,37.169,-50.008,-179.890,6.283,149.106
C07953=1149.311,36.920,-49.993,-179.894,6.282,149.106
C07954=1149.316,36.670,-49.978,-179.896,6.281,149.107
C07955=1149.321,36.420,-49.963,-179.898,6.281,149.108
C07956=1149.326,36.170,-49.948,-179.901,6.279,149.108
C07957=1149.331,35.921,-49.933,-179.904,6.278,149.109
C07958=1149.336,35.672,-49.918,-179.907,6.277,149.109
C07959=1149.341,35.422,-49.903,-179.909,6.276,149.110
C07960=1149.346,35.173,-49.888,-179.911,6.276,149.110
C07961=1149.351,34.923,-49.874,-179.914,6.274,149.111
C07962=1149.356,34.674,-49.858,-179.917,6.273,149.111
C07963=1149.361,34.424,-49.844,-179.919,6.273,149.112
C07964=1149.366,34.175,-49.829,-179.922,6.271,149.113
C07965=1149.372,33.925,-49.814,-179.924,6.271,149.113
C07966=1149.376,33.676,-49.799,-179.927,6.269,149.113
C07967=1149.381,33.426,-49.785,-179.930,6.268,149.114
C07968=1149.387,33.177,-49.769,-179.932,6.268,149.115
C07969=1149.392,32.927,-49.755,-179.935,6.266,149.115
C07970=1149.396,32.678,-49.740,-179.937,6.265,149.116
C07971=1149.402,32.428,-49.725,-179.940,6.265,149.116
C07972=1149.407,32.178,-49.711,-179.943,6.263,149.117
C07973=1149.411,31.929,-49.696,-179.945,6.263,149.117
C07974=1149.417,31.679,-49.681,-179.948,6.262,149.118
C07975=1149.422,31.430,-49.666,-179.950,6.260,149.118
C07976=1149.427,31.181,-49.652,-179.953,6.260,149.119
C07977=1149.432,30.932,-49.637,-179.955,6.259,149.120
C07978=1149.438,30.682,-49.622,-179.958,6.258,149.120
C07979=1149.443,30.432,-49.608,-179.961,6.257,149.121
C07980=1149.447,30.183,-49.593,-179.963,6.256,149.121
C07981=1149.452,29.934,-49.578,-179.966,6.255,149.122
C07982=1149.458,29.684,-49.563,-179.968,6.254,149.122
C07983=1149.463,29.435,-49.548,-179.971,6.253,149.123
C07984=1149.468,29.185,-49.534,-179.973,6.252,149.123
C07985=1149.473,28.935,-49.520,-179.976,6.252,149.124
C07986=1149.477,28.686,-49.505,-179.979,6.250,149.125
C07987=1149.483,28.436,-49.490,-179.981,6.249,149.125
C07988=1149.488,28.186,-49.476,-179.984,6.249,149.126
C07989=1149.493,27.917,-49.460,-179.987,6.247,149.126
C07990=1149.499,27.649,-49.445,-179.989,6.247,149.127
C07991=1149.505,27.380,-49.429,-179.992,6.245,149.127
C07992=1149.510,27.111,-49.413,-179.995,6.244,149.128
C07993=1149.515,26.861,-49.399,-179.998,6.243,149.129
C07994=1149.520,26.612,-49.384,-180.000,6.242,149.129
C07995=1149.525,26.362,-49.370,179.997,6.242,149.130
C07996=1149.530,26.112,-49.355,179.995,6.241,149.130
C07997=1149.535,25.863,-49.341,179.992,6.240,149.131
C07998=1149.540,25.614,-49.326,179.990,6.239,149.131
C07999=1149.545,25.365,-49.312,179.987,6.239,149.132
C08000=1149.550,25.115,-49.298,179.984,6.237,149.132
C08001=1149.555,24.865,-49.283,179.982,6.236,149.133
C08002=1149.560,24.615,-49.269,179.980,6.236,149.134
C08003=1149.565,24.366,-49.255,179.977,6.234,149.134
C08004=1149.570,24.117,-49.240,179.974,6.234,149.135
C08005=1149.575,23.868,-49.226,179.972,6.233,149.135
C08006=1149.581,23.618,-49.211,179.969,6.231,149.136
C08007=1149.586,23.368,-49.197,179.967,6.231,149.136
C08008=1149.591,23.118,-49.182,179.964,6.230,149.137
C08009=1149.596,22.868,-49.168,179.962,6.229,149.137
C08010=1149.601,22.619,-49.154,179.959,6.228,149.138
C08011=1149.606,22.370,-49.140,179.956,6.227,149.139
C08012=1149.611,22.120,-49.126,179.954,6.226,149.139
C08013=1149.616,21.870,-49.111,179.951,6.225,149.140
C08014=1149.621,21.621,-49.097,179.949,6.224,149.140
C08015=1149.627,21.372,-49.083,179.946,6.224,149.141
C08016=1149.632,21.122,-49.068,179.944,6.223,149.141
C08017=1149.636,20.873,-49.054,179.941,6.222,149.142
C08018=1149.641,20.623,-49.040,179.939,6.221,149.142
C08019=1149.646,20.373,-49.025,179.936,6.220,149.143
C08020=1149.652,20.124,-49.011,179.933,6.219,149.144
C08021=1149.657,19.875,-48.997,179.931,6.218,149.144
C08022=1149.662,19.625,-48.983,179.928,6.218,149.145
C08023=1149.667,19.375,-48.969,179.926,6.217,149.145
C08024=1149.673,19.126,-48.955,179.923,6.216,149.146
C08025=1149.678,18.876,-48.941,179.921,6.215,149.146
C08026=1149.683,18.626,-48.927,179.918,6.214,149.147
C08027=1149.688,18.376,-48.913,179.916,6.213,149.147
C08028=1149.693,18.127,-48.899,179.913,6.212,149.148
C08029=1149.697,17.878,-48.885,179.911,6.211,149.149
C08030=1149.702,17.628,-48.871,179.908,6.211,149.149
C08031=1149.708,17.379,-48.857,179.905,6.209,149.150
C08032=1149.713,17.130,-48.843,179.903,6.208,149.150
C08033=1149.718,16.880,-48.828,179.900,6.208,149.151
C08034=1149.723,16.630,-48.814,179.898,6.207,149.151
C08035=1149.729,16.381,-48.801,179.895,6.206,149.152
C08036=1149.733,16.131,-48.786,179.893,6.205,149.152
C08037=1149.738,15.881,-48.772,179.890,6.205,149.153
C08038=1149.744,15.632,-48.758,179.888,6.204,149.154
C08039=1149.748,15.383,-48.745,179.885,6.202,149.154
C08040=1149.753,15.133,-48.730,179.882,6.202,149.155
C08041=1149.759,14.883,-48.717,179.880,6.201,149.155
C08042=1149.764,14.634,-48.703,179.878,6.200,149.156
C08043=1149.769,14.384,-48.689,179.875,6.200,149.156
C08044=1149.774,14.134,-48.674,179.872,6.198,149.157
C08045=1149.779,13.885,-48.660,179.870,6.198,149.157
C08046=1149.784,13.635,-48.647,179.867,6.197,149.158
C08047=1149.790,13.386,-48.634,179.865,6.196,149.159
C08048=1149.794,13.137,-48.619,179.862,6.195,149.159
C08049=1149.799,12.887,-48.605,179.860,6.194,149.160
C08050=1149.805,12.637,-48.592,179.858,6.193,149.160
C08051=1149.810,12.388,-48.578,179.855,6.193,149.161
C08052=1149.814,12.138,-48.564,179.852,6.191,149.161
C08053=1149.820,11.888,-48.551,179.850,6.191,149.162
C08054=1149.825,11.639,-48.536,179.847,6.190,149.163
C08055=1149.830,11.389,-48.523,179.845,6.190,149.163
C08056=1149.835,11.140,-48.509,179.843,6.189,149.164
C08057=1149.840,10.890,-48.495,179.839,6.188,149.164
C08058=1149.846,10.641,-48.481,179.837,6.187,149.165
C08059=1149.850,10.392,-48.468,179.835,6.186,149.165
C08060=1149.855,10.141,-48.454,179.832,6.185,149.166
C08061=1149.861,9.892,-48.440,179.829,6.184,149.167
C08062=1149.866,9.642,-48.427,179.827,6.183,149.167
C08063=1149.871,9.393,-48.413,179.825,6.183,149.168
C08064=1149.876,9.144,-48.399,179.822,6.182,149.168
C08065=1149.881,8.893,-48.385,179.820,6.181,149.169
C08066=1149.887,8.644,-48.371,179.817,6.180,149.169
C08067=1149.891,8.394,-48.359,179.815,6.179,149.170
C08068=1149.897,8.145,-48.345,179.812,6.179,149.171
C08069=1149.902,7.895,-48.330,179.810,6.178,149.171
C08070=1149.907,7.646,-48.318,179.807,6.178,149.172
C08071=1149.912,7.396,-48.303,179.804,6.176,149.172
C08072=1149.917,7.146,-48.290,179.802,6.176,149.173
C08073=1149.922,6.897,-48.277,179.799,6.175,149.173
C08074=1149.927,6.647,-48.263,179.797,6.174,149.174
C08075=1149.933,6.398,-48.249,179.795,6.173,149.174
C08076=1149.937,6.148,-48.236,179.792,6.172,149.175
C08077=1149.943,5.899,-48.222,179.789,6.171,149.176
C08078=1149.947,5.649,-48.209,179.787,6.171,149.176
C08079=1149.953,5.400,-48.195,179.784,6.170,149.177
C08080=1149.958,5.150,-48.182,179.782,6.169,149.177
C08081=1149.963,4.901,-48.168,179.780,6.169,149.178
C08082=1149.968,4.651,-48.155,179.777,6.167,149.178
C08083=1149.973,4.402,-48.142,179.774,6.167,149.179
C08084=1149.978,4.152,-48.128,179.772,6.166,149.180
C08085=1149.984,3.902,-48.115,179.769,6.166,149.180
C08086=1149.988,3.653,-48.101,179.767,6.165,149.181
C08087=1149.994,3.403,-48.088,179.764,6.164,149.181
C08088=1149.999,3.154,-48.074,179.762,6.163,149.182
C08089=1150.004,2.904,-48.061,179.760,6.162,149.182
C08090=1150.009,2.654,-48.048,179.757,6.161,149.183
C08091=1150.014,2.405,-48.034,179.755,6.161,149.183
C08092=1150.020,2.155,-48.021,179.752,6.160,149.184
C08093=1150.025,1.886,-48.007,179.749,6.159,149.185
C08094=1150.031,1.616,-47.992,179.747,6.158,149.185
C08095=1150.036,1.347,-47.977,179.744,6.158,149.186
C08096=1150.041,1.077,-47.964,179.741,6.156,149.187
C08097=1150.047,0.828,-47.950,179.739,6.156,149.187
C08098=1150.051,0.578,-47.937,179.736,6.155,149.188
C08099=1150.057,0.328,-47.924,179.734,6.154,149.188
C08100=1150.062,0.080,-47.910,179.732,6.154,149.189
C08101=1150.067,-0.171,-47.897,179.729,6.153,149.189
C08102=1150.072,-0.420,-47.884,179.726,6.151,149.190
C08103=1150.078,-0.670,-47.871,179.723,6.151,149.191
C08104=1150.082,-0.919,-47.857,179.721,6.150,149.191
C08105=1150.088,-1.169,-47.844,179.719,6.150,149.192
C08106=1150.093,-1.419,-47.831,179.716,6.149,149.192
C08107=1150.099,-1.668,-47.818,179.714,6.149,149.193
C08108=1150.103,-1.918,-47.804,179.712,6.148,149.193
C08109=1150.109,-2.167,-47.791,179.709,6.147,149.194
C08110=1150.113,-2.417,-47.778,179.706,6.146,149.194
C08111=1150.118,-2.667,-47.765,179.704,6.145,149.195
C08112=1150.124,-2.916,-47.752,179.701,6.144,149.196
C08113=1150.128,-3.166,-47.739,179.699,6.144,149.196
C08114=1150.134,-3.415,-47.725,179.696,6.143,149.197
C08115=1150.139,-3.665,-47.713,179.694,6.142,149.197
C08116=1150.145,-3.915,-47.699,179.692,6.142,149.198
C08117=1150.150,-4.164,-47.687,179.689,6.140,149.198
C08118=1150.154,-4.414,-47.674,179.686,6.140,149.199
C08119=1150.160,-4.663,-47.660,179.684,6.139,149.200
C08120=1150.165,-4.913,-47.647,179.681,6.139,149.200
C08121=1150.170,-5.163,-47.634,179.679,6.138,149.201
C08122=1150.175,-5.412,-47.621,179.677,6.137,149.201
C08123=1150.181,-5.662,-47.608,179.674,6.137,149.202
C08124=1150.185,-5.912,-47.595,179.672,6.136,149.203
C08125=1150.191,-6.161,-47.582,179.670,6.135,149.203
C08126=1150.196,-6.411,-47.570,179.667,6.134,149.204
C08127=1150.201,-6.661,-47.557,179.664,6.133,149.204
C08128=1150.206,-6.910,-47.543,179.662,6.133,149.205
C08129=1150.212,-7.160,-47.531,179.659,6.132,149.205
C08130=1150.216,-7.410,-47.518,179.657,6.131,149.206
C08131=1150.222,-7.659,-47.505,179.654,6.131,149.207
C08132=1150.227,-7.908,-47.491,179.652,6.130,149.207
C08133=1150.231,-8.158,-47.478,179.650,6.130,149.208
C08134=1150.237,-8.408,-47.465,179.647,6.129,149.208
C08135=1150.242,-8.657,-47.453,179.645,6.128,149.209
C08136=1150.247,-8.907,-47.440,179.642,6.127,149.209
C08137=1150.252,-9.156,-47.427,179.639,6.126,149.210
C08138=1150.258,-9.406,-47.414,179.637,6.126,149.210
C08139=1150.263,-9.656,-47.402,179.635,6.125,149.211
C08140=1150.268,-9.906,-47.389,179.632,6.124,149.212
C08141=1150.273,-10.155,-47.376,179.630,6.123,149.212
C08142=1150.279,-10.405,-47.363,179.628,6.123,149.213
C08143=1150.284,-10.654,-47.351,179.625,6.122,149.213
C08144=1150.288,-10.904,-47.338,179.623,6.122,149.214
C08145=1150.293,-11.153,-47.325,179.620,6.121,149.214
C08146=1150.299,-11.403,-47.312,179.618,6.121,149.215
C08147=1150.304,-11.653,-47.299,179.615,6.119,149.216
C08148=1150.309,-11.902,-47.286,179.612,6.119,149.216
C08149=1150.314,-12.152,-47.274,179.610,6.118,149.217
C08150=1150.319,-12.401,-47.261,179.608,6.117,149.217
C08151=1150.325,-12.652,-47.248,179.605,6.116,149.218
C08152=1150.330,-12.901,-47.236,179.603,6.116,149.219
C08153=1150.335,-13.151,-47.223,179.601,6.115,149.219
C08154=1150.340,-13.400,-47.210,179.598,6.115,149.220
C08155=1150.345,-13.649,-47.198,179.596,6.114,149.220
C08156=1150.350,-13.899,-47.185,179.594,6.113,149.221
C08157=1150.356,-14.149,-47.172,179.591,6.113,149.221
C08158=1150.361,-14.399,-47.160,179.589,6.112,149.222
C08159=1150.366,-14.648,-47.147,179.586,6.112,149.223
C08160=1150.371,-14.897,-47.135,179.584,6.111,149.223
C08161=1150.376,-15.147,-47.122,179.581,6.110,149.224
C08162=1150.381,-15.397,-47.110,179.578,6.109,149.224
C08163=1150.386,-15.647,-47.097,179.576,6.108,149.225
C08164=1150.392,-15.896,-47.084,179.574,6.107,149.225
C08165=1150.397,-16.146,-47.071,179.571,6.107,149.226
C08166=1150.402,-16.396,-47.059,179.569,6.106,149.226
C08167=1150.407,-16.646,-47.046,179.566,6.106,149.227
C08168=1150.412,-16.895,-47.034,179.564,6.105,149.228
C08169=1150.418,-17.144,-47.021,179.562,6.104,149.228
C08170=1150.423,-17.394,-47.009,179.559,6.104,149.229
C08171=1150.428,-17.643,-46.997,179.557,6.103,149.229
C08172=1150.433,-17.894,-46.984,179.554,6.103,149.230
C08173=1150.438,-18.143,-46.972,179.552,6.102,149.230
C08174=1150.443,-18.393,-46.959,179.549,6.101,149.231
C08175=1150.448,-18.642,-46.947,179.547,6.101,149.232
C08176=1150.454,-18.892,-46.935,179.545,6.100,149.232
C08177=1150.459,-19.141,-46.922,179.542,6.099,149.233
C08178=1150.464,-19.391,-46.910,179.540,6.099,149.233
C08179=1150.469,-19.641,-46.898,179.538,6.098,149.234
C08180=1150.474,-19.891,-46.885,179.535,6.098,149.235
C08181=1150.480,-20.140,-46.872,179.533,6.097,149.235
C08182=1150.485,-20.390,-46.860,179.531,6.096,149.236
C08183=1150.490,-20.640,-46.847,179.528,6.096,149.236
C08184=1150.496,-20.889,-46.835,179.526,6.095,149.237
C08185=1150.501,-21.139,-46.823,179.523,6.094,149.237
C08186=1150.506,-21.388,-46.810,179.521,6.094,149.238
C08187=1150.512,-21.638,-46.798,179.518,6.093,149.239
C08188=1150.516,-21.887,-46.786,179.516,6.092,149.239
C08189=1150.521,-22.137,-46.774,179.513,6.092,149.240
C08190=1150.526,-22.387,-46.761,179.511,6.091,149.240
C08191=1150.531,-22.637,-46.749,179.508,6.091,149.241
C08192=1150.536,-22.886,-46.737,179.506,6.090,149.241
C08193=1150.542,-23.136,-46.725,179.504,6.090,149.242
C08194=1150.547,-23.385,-46.712,179.501,6.089,149.243
C08195=1150.552,-23.635,-46.700,179.499,6.087,149.243
C08196=1150.558,-23.885,-46.688,179.496,6.087,149.244
C08197=1150.563,-24.155,-46.675,179.493,6.086,149.244
C08198=1150.569,-24.424,-46.661,179.491,6.086,149.245
C08199=1150.574,-24.695,-46.648,179.488,6.085,149.246
C08200=1150.580,-24.964,-46.635,179.486,6.085,149.246
C08201=1150.585,-25.214,-46.622,179.484,6.084,149.247
C08202=1150.590,-25.464,-46.611,179.481,6.083,149.247
C08203=1150.595,-25.714,-46.598,179.479,6.083,149.248
C08204=1150.601,-25.964,-46.586,179.477,6.082,149.248
C08205=1150.606,-26.213,-46.575,179.474,6.081,149.249
C08206=1150.611,-26.463,-46.562,179.472,6.081,149.250
C08207=1150.616,-26.713,-46.550,179.469,6.080,149.250
C08208=1150.621,-26.962,-46.538,179.467,6.079,149.251
C08209=1150.627,-27.212,-46.526,179.464,6.079,149.251
C08210=1150.632,-27.462,-46.514,179.462,6.078,149.252
C08211=1150.637,-27.711,-46.501,179.459,6.078,149.253
C08212=1150.642,-27.961,-46.490,179.457,6.077,149.253
C08213=1150.647,-28.211,-46.478,179.455,6.076,149.254
C08214=1150.652,-28.460,-46.465,179.452,6.076,149.254
C08215=1150.658,-28.710,-46.454,179.450,6.075,149.255
C08216=1150.663,-28.959,-46.441,179.448,6.075,149.255
C08217=1150.668,-29.209,-46.430,179.445,6.074,149.256
C08218=1150.673,-29.459,-46.418,179.443,6.073,149.257
C08219=1150.678,-29.708,-46.405,179.441,6.073,149.257
C08220=1150.684,-29.958,-46.393,179.438,6.072,149.258
C08221=1150.689,-30.208,-46.381,179.436,6.071,149.258
C08222=1150.694,-30.458,-46.370,179.433,6.071,149.259
C08223=1150.699,-30.707,-46.358,179.431,6.070,149.259
C08224=1150.705,-30.956,-46.346,179.429,6.069,149.260
C08225=1150.710,-31.206,-46.334,179.426,6.069,149.261
C08226=1150.715,-31.456,-46.323,179.424,6.068,149.261
C08227=1150.720,-31.705,-46.310,179.421,6.068,149.262
C08228=1150.726,-31.955,-46.298,179.419,6.067,149.262
C08229=1150.731,-32.205,-46.287,179.416,6.067,149.263
C08230=1150.736,-32.454,-46.275,179.415,6.067,149.263
C08231=1150.741,-32.704,-46.263,179.412,6.066,149.264
C08232=1150.746,-32.954,-46.251,179.410,6.065,149.265
C08233=1150.752,-33.204,-46.239,179.408,6.064,149.265
C08234=1150.756,-33.453,-46.228,179.405,6.064,149.266
C08235=1150.762,-33.703,-46.216,179.403,6.063,149.266
C08236=1150.767,-33.953,-46.203,179.400,6.063,149.267
C08237=1150.772,-34.201,-46.192,179.398,6.062,149.267
C08238=1150.778,-34.451,-46.180,179.395,6.062,149.268
C08239=1150.783,-34.701,-46.168,179.393,6.061,149.269
C08240=1150.788,-34.951,-46.157,179.390,6.060,149.269
C08241=1150.793,-35.201,-46.145,179.388,6.060,149.270
C08242=1150.798,-35.450,-46.133,179.386,6.059,149.270
C08243=1150.803,-35.700,-46.121,179.383,6.058,149.271
C08244=1150.809,-35.950,-46.109,179.381,6.058,149.271
C08245=1150.814,-36.200,-46.098,179.379,6.057,149.272
C08246=1150.819,-36.449,-46.087,179.376,6.056,149.273
C08247=1150.825,-36.699,-46.075,179.374,6.056,149.273
C08248=1150.830,-36.949,-46.063,179.372,6.056,149.274
C08249=1150.835,-37.198,-46.052,179.369,6.056,149.274
C08250=1150.840,-37.448,-46.040,179.367,6.055,149.275
C08251=1150.846,-37.698,-46.028,179.365,6.054,149.275
C08252=1150.850,-37.948,-46.016,179.362,6.054,149.276
C08253=1150.856,-38.197,-46.005,179.360,6.053,149.277
C08254=1150.861,-38.446,-45.994,179.358,6.052,149.277
C08255=1150.866,-38.696,-45.981,179.355,6.052,149.278
C08256=1150.872,-38.946,-45.969,179.353,6.051,149.278
C08257=1150.876,-39.195,-45.958,179.351,6.050,149.279
C08258=1150.882,-39.445,-45.946,179.348,6.050,149.280
C08259=1150.887,-39.694,-45.935,179.346,6.049,149.280
C08260=1150.892,-39.944,-45.923,179.344,6.049,149.281
C08261=1150.898,-40.194,-45.911,179.341,6.049,149.281
C08262=1150.903,-40.444,-45.900,179.339,6.048,149.282
C08263=1150.908,-40.694,-45.889,179.337,6.048,149.282
C08264=1150.914,-40.943,-45.878,179.334,6.047,149.283
C08265=1150.919,-41.193,-45.866,179.332,6.046,149.284
C08266=1150.924,-41.443,-45.855,179.330,6.046,149.284
C08267=1150.929,-41.693,-45.843,179.327,6.045,149.285
C08268=1150.934,-41.942,-45.832,179.325,6.044,149.285
C08269=1150.940,-42.192,-45.820,179.323,6.044,149.286
C08270=1150.945,-42.441,-45.809,179.320,6.043,149.286
C08271=1150.950,-42.691,-45.797,179.318,6.043,149.287
C08272=1150.955,-42.941,-45.786,179.316,6.043,149.288
C08273=1150.961,-43.190,-45.774,179.313,6.042,149.288
C08274=1150.965,-43.440,-45.763,179.311,6.042,149.289
C08275=1150.971,-43.690,-45.751,179.309,6.041,149.289
C08276=1150.976,-43.940,-45.740,179.306,6.040,149.290
C08277=1150.982,-44.189,-45.729,179.304,6.040,149.290
C08278=1150.987,-44.439,-45.718,179.302,6.039,149.291
C08279=1150.992,-44.689,-45.706,179.299,6.039,149.292
C08280=1150.997,-44.938,-45.694,179.297,6.039,149.292
C08281=1151.003,-45.187,-45.683,179.295,6.038,149.293
C08282=1151.008,-45.438,-45.672,179.292,6.037,149.293
C08283=1151.012,-45.687,-45.661,179.290,6.037,149.294
C08284=1151.018,-45.937,-45.649,179.288,6.036,149.294
C08285=1151.023,-46.186,-45.638,179.285,6.035,149.295
C08286=1151.029,-46.436,-45.626,179.283,6.035,149.296
C08287=1151.034,-46.686,-45.616,179.281,6.034,149.296
C08288=1151.040,-46.936,-45.604,179.278,6.034,149.297
C08289=1151.044,-47.185,-45.593,179.276,6.034,149.297
C08290=1151.049,-47.435,-45.582,179.274,6.033,149.298
C08291=1151.055,-47.685,-45.570,179.271,6.033,149.298
C08292=1151.060,-47.934,-45.560,179.269,6.032,149.299
C08293=1151.065,-48.184,-45.548,179.267,6.031,149.300
C08294=1151.070,-48.434,-45.536,179.264,6.031,149.300
C08295=1151.076,-48.683,-45.526,179.262,6.030,149.301
C08296=1151.081,-48.933,-45.514,179.260,6.030,149.301
C08297=1151.086,-49.183,-45.503,179.258,6.029,149.302
C08298=1151.091,-49.432,-45.492,179.255,6.029,149.303
C08299=1151.097,-49.682,-45.481,179.253,6.028,149.303
C08300=1151.102,-49.932,-45.470,179.250,6.028,149.304
C08301=1151.108,-50.202,-45.458,179.248,6.027,149.304
C08302=1151.113,-50.473,-45.445,179.246,6.027,149.305
C08303=1151.119,-50.744,-45.433,179.243,6.026,149.305
C08304=1151.125,-51.015,-45.421,179.241,6.025,149.306
C08305=1151.130,-51.264,-45.410,179.239,6.025,149.307
C08306=1151.135,-51.515,-45.399,179.236,6.024,149.307
C08307=1151.140,-51.763,-45.389,179.234,6.024,149.308
C08308=1151.146,-52.013,-45.377,179.232,6.024,149.308
C08309=1151.151,-52.263,-45.366,179.229,6.023,149.309
C08310=1151.156,-52.513,-45.355,179.227,6.023,149.310
C08311=1151.161,-52.762,-45.343,179.225,6.022,149.310
C08312=1151.167,-53.012,-45.333,179.222,6.021,149.311
C08313=1151.172,-53.262,-45.322,179.220,6.021,149.311
C08314=1151.177,-53.512,-45.311,179.218,6.021,149.312
C08315=1151.183,-53.761,-45.300,179.215,6.020,149.312
C08316=1151.188,-54.011,-45.289,179.213,6.020,149.313
C08317=1151.193,-54.260,-45.278,179.211,6.019,149.313
C08318=1151.198,-54.510,-45.267,179.208,6.018,149.314
C08319=1151.203,-54.760,-45.256,179.206,6.018,149.315
C08320=1151.209,-55.009,-45.245,179.204,6.018,149.315
C08321=1151.214,-55.260,-45.234,179.202,6.017,149.316
C08322=1151.219,-55.509,-45.223,179.200,6.016,149.316
C08323=1151.225,-55.759,-45.212,179.197,6.016,149.317
C08324=1151.229,-56.009,-45.201,179.195,6.015,149.317
C08325=1151.235,-56.258,-45.191,179.192,6.015,149.318
C08326=1151.240,-56.508,-45.179,179.191,6.015,149.319
C08327=1151.245,-56.757,-45.169,179.188,6.014,149.319
C08328=1151.251,-57.007,-45.157,179.186,6.014,149.320
C08329=1151.256,-57.257,-45.147,179.184,6.013,149.320
C08330=1151.261,-57.507,-45.136,179.181,6.013,149.321
C08331=1151.266,-57.757,-45.125,179.179,6.012,149.321
C08332=1151.271,-58.006,-45.114,179.177,6.012,149.322
C08333=1151.276,-58.256,-45.104,179.174,6.011,149.323
C08334=1151.283,-58.506,-45.093,179.172,6.011,149.323
C08335=1151.287,-58.755,-45.082,179.170,6.010,149.324
C08336=1151.293,-59.005,-45.071,179.167,6.009,149.324
C08337=1151.298,-59.255,-45.060,179.166,6.009,149.325
C08338=1151.303,-59.504,-45.050,179.163,6.009,149.325
C08339=1151.308,-59.754,-45.039,179.161,6.008,149.326
C08340=1151.313,-60.004,-45.028,179.158,6.008,149.327
C08341=1151.319,-60.254,-45.018,179.156,6.007,149.327
C08342=1151.324,-60.504,-45.006,179.155,6.007,149.328
C08343=1151.330,-60.753,-44.996,179.152,6.007,149.328
C08344=1151.335,-61.003,-44.985,179.150,6.006,149.329
C08345=1151.340,-61.252,-44.974,179.147,6.006,149.330
C08346=1151.345,-61.502,-44.964,179.145,6.005,149.330
C08347=1151.350,-61.752,-44.953,179.143,6.005,149.330
C08348=1151.355,-62.002,-44.942,179.141,6.004,149.331
C08349=1151.361,-62.251,-44.932,179.138,6.004,149.332
C08350=1151.366,-62.501,-44.921,179.136,6.003,149.332
C08351=1151.371,-62.750,-44.910,179.134,6.002,149.333
C08352=1151.376,-63.001,-44.900,179.132,6.002,149.333
C08353=1151.382,-63.250,-44.889,179.129,6.002,149.334
C08354=1151.387,-63.500,-44.878,179.127,6.001,149.335
C08355=1151.393,-63.750,-44.868,179.124,6.001,149.335
C08356=1151.398,-63.999,-44.857,179.122,6.000,149.336
C08357=1151.403,-64.249,-44.847,179.121,6.000,149.336
C08358=1151.409,-64.498,-44.836,179.118,6.000,149.337
C08359=1151.414,-64.749,-44.825,179.116,5.999,149.337
C08360=1151.419,-64.998,-44.815,179.114,5.998,149.338
C08361=1151.424,-65.248,-44.804,179.112,5.999,149.339
C08362=1151.429,-65.497,-44.794,179.109,5.998,149.339
C08363=1151.434,-65.748,-44.783,179.107,5.997,149.340
C08364=1151.440,-65.997,-44.773,179.104,5.997,149.340
C08365=1151.445,-66.247,-44.762,179.102,5.996,149.341
C08366=1151.451,-66.497,-44.752,179.100,5.996,149.341
C08367=1151.456,-66.746,-44.741,179.098,5.995,149.342
C08368=1151.461,-66.996,-44.730,179.096,5.995,149.342
C08369=1151.466,-67.246,-44.720,179.093,5.994,149.343
C08370=1151.471,-67.496,-44.710,179.092,5.994,149.344
C08371=1151.477,-67.745,-44.699,179.089,5.994,149.344
C08372=1151.483,-67.995,-44.689,179.087,5.993,149.345
C08373=1151.487,-68.245,-44.678,179.084,5.992,149.345
C08374=1151.493,-68.494,-44.668,179.082,5.993,149.346
C08375=1151.498,-68.744,-44.657,179.080,5.992,149.346
C08376=1151.504,-68.994,-44.647,179.078,5.991,149.347
C08377=1151.509,-69.243,-44.637,179.075,5.991,149.348
C08378=1151.513,-69.493,-44.627,179.074,5.991,149.348
C08379=1151.519,-69.743,-44.617,179.071,5.990,149.349
C08380=1151.524,-69.993,-44.606,179.069,5.990,149.349
C08381=1151.530,-70.243,-44.596,179.067,5.989,149.350
C08382=1151.535,-70.492,-44.585,179.065,5.989,149.350
C08383=1151.540,-70.742,-44.574,179.062,5.989,149.351
C08384=1151.546,-70.991,-44.564,179.060,5.988,149.351
C08385=1151.551,-71.241,-44.554,179.058,5.987,149.352
C08386=1151.556,-71.491,-44.543,179.056,5.987,149.353
C08387=1151.562,-71.741,-44.533,179.054,5.987,149.353
C08388=1151.567,-71.991,-44.523,179.051,5.986,149.354
C08389=1151.572,-72.241,-44.512,179.049,5.985,149.354
C08390=1151.577,-72.490,-44.503,179.047,5.986,149.355
C08391=1151.582,-72.740,-44.492,179.045,5.985,149.355
C08392=1151.588,-72.990,-44.482,179.043,5.984,149.356
C08393=1151.593,-73.239,-44.472,179.040,5.984,149.357
C08394=1151.598,-73.489,-44.461,179.038,5.984,149.357
C08395=1151.604,-73.739,-44.451,179.036,5.983,149.358
C08396=1151.610,-73.988,-44.441,179.033,5.983,149.358
C08397=1151.614,-74.238,-44.431,179.031,5.982,149.359
C08398=1151.619,-74.488,-44.421,179.030,5.982,149.359
C08399=1151.625,-74.737,-44.410,179.027,5.982,149.360
C08400=1151.631,-74.987,-44.400,179.025,5.981,149.360
C08401=1151.636,-75.237,-44.390,179.023,5.980,149.361
C08402=1151.641,-75.487,-44.379,179.020,5.981,149.362
C08403=1151.646,-75.736,-44.370,179.018,5.980,149.362
C08404=1151.651,-75.986,-44.359,179.016,5.979,149.363
C08405=1151.658,-76.258,-44.349,179.013,5.979,149.363
C08406=1151.663,-76.529,-44.338,179.011,5.979,149.364
C08407=1151.669,-76.801,-44.326,179.009,5.978,149.365
C08408=1151.675,-77.071,-44.316,179.006,5.978,149.365
C08409=1151.680,-77.321,-44.305,179.004,5.977,149.366
C08410=1151.685,-77.571,-44.295,179.002,5.976,149.366
C08411=1151.690,-77.820,-44.285,179.000,5.977,149.367
C08412=1151.696,-78.070,-44.276,178.998,5.976,149.367
C08413=1151.701,-78.321,-44.265,178.996,5.975,149.368
C08414=1151.707,-78.570,-44.255,178.993,5.975,149.369
C08415=1151.712,-78.820,-44.245,178.991,5.975,149.369
C08416=1151.717,-79.069,-44.235,178.989,5.974,149.370
C08417=1151.722,-79.319,-44.225,178.986,5.974,149.370
C08418=1151.728,-79.569,-44.215,178.985,5.974,149.371
C08419=1151.733,-79.819,-44.205,178.983,5.973,149.371
C08420=1151.739,-80.068,-44.195,178.980,5.973,149.372
C08421=1151.744,-80.318,-44.185,178.978,5.973,149.372
C08422=1151.749,-80.568,-44.174,178.976,5.972,149.373
C08423=1151.754,-80.818,-44.166,178.974,5.971,149.374
C08424=1151.760,-81.067,-44.155,178.971,5.971,149.374
C08425=1151.765,-81.318,-44.145,178.970,5.971,149.375
C08426=1151.770,-81.567,-44.135,178.967,5.970,149.375
C08427=1151.775,-81.816,-44.125,178.965,5.970,149.376
C08428=1151.781,-82.067,-44.115,178.963,5.970,149.376
C08429=1151.786,-82.316,-44.106,178.961,5.969,149.377
C08430=1151.791,-82.566,-44.095,178.958,5.968,149.377
C08431=1151.797,-82.816,-44.085,178.957,5.968,149.378
C08432=1151.802,-83.065,-44.076,178.954,5.968,149.379
C08433=1151.808,-83.315,-44.066,178.952,5.967,149.379
C08434=1151.813,-83.564,-44.056,178.950,5.967,149.380
C08435=1151.818,-83.815,-44.047,178.948,5.967,149.380
C08436=1151.823,-84.065,-44.036,178.946,5.966,149.381
C08437=1151.829,-84.314,-44.026,178.943,5.965,149.381
C08438=1151.834,-84.564,-44.017,178.941,5.966,149.382
C08439=1151.840,-84.814,-44.007,178.939,5.965,149.382
C08440=1151.844,-85.063,-43.997,178.937,5.964,149.383
C08441=1151.849,-85.313,-43.987,178.935,5.965,149.384
C08442=1151.855,-85.563,-43.977,178.933,5.964,149.384
C08443=1151.860,-85.812,-43.968,178.930,5.963,149.385
C08444=1151.866,-86.063,-43.958,178.929,5.963,149.385
C08445=1151.871,-86.312,-43.949,178.926,5.963,149.386
C08446=1151.876,-86.562,-43.938,178.924,5.962,149.386
C08447=1151.882,-86.812,-43.929,178.922,5.962,149.387
C08448=1151.887,-87.061,-43.919,178.920,5.962,149.388
C08449=1151.892,-87.311,-43.909,178.918,5.961,149.388
C08450=1151.898,-87.561,-43.900,178.916,5.961,149.388
C08451=1151.903,-87.810,-43.890,178.913,5.961,149.389
C08452=1151.908,-88.061,-43.880,178.911,5.960,149.390
C08453=1151.913,-88.310,-43.870,178.909,5.960,149.390
C08454=1151.919,-88.560,-43.860,178.907,5.959,149.391
C08455=1151.924,-88.810,-43.851,178.905,5.959,149.391
C08456=1151.930,-89.059,-43.841,178.903,5.959,149.392
C08457=1151.935,-89.309,-43.832,178.901,5.958,149.392
C08458=1151.940,-89.559,-43.822,178.898,5.958,149.393
C08459=1151.946,-89.809,-43.813,178.897,5.958,149.393
C08460=1151.951,-90.059,-43.802,178.894,5.957,149.394
C08461=1151.956,-90.309,-43.793,178.892,5.956,149.395
C08462=1151.961,-90.558,-43.783,178.890,5.956,149.395
C08463=1151.967,-90.808,-43.774,178.888,5.956,149.396
C08464=1151.972,-91.058,-43.764,178.886,5.955,149.396
C08465=1151.977,-91.308,-43.755,178.884,5.955,149.397
C08466=1151.983,-91.557,-43.745,178.881,5.955,149.397
C08467=1151.988,-91.807,-43.736,178.879,5.954,149.398
C08468=1151.994,-92.056,-43.726,178.877,5.954,149.399
C08469=1151.999,-92.306,-43.717,178.875,5.954,149.399
C08470=1152.004,-92.556,-43.707,178.873,5.953,149.400
C08471=1152.010,-92.806,-43.698,178.871,5.953,149.400
C08472=1152.015,-93.056,-43.687,178.868,5.952,149.401
C08473=1152.020,-93.306,-43.678,178.867,5.952,149.401
C08474=1152.025,-93.555,-43.669,178.865,5.952,149.402
C08475=1152.031,-93.805,-43.659,178.862,5.951,149.402
C08476=1152.035,-94.054,-43.650,178.860,5.951,149.403
C08477=1152.041,-94.305,-43.640,178.858,5.951,149.403
C08478=1152.046,-94.554,-43.631,178.856,5.950,149.404
C08479=1152.052,-94.804,-43.621,178.854,5.950,149.405
C08480=1152.057,-95.054,-43.612,178.852,5.949,149.405
C08481=1152.063,-95.303,-43.602,178.850,5.949,149.406
C08482=1152.068,-95.553,-43.593,178.847,5.949,149.406
C08483=1152.073,-95.803,-43.584,178.845,5.948,149.407
C08484=1152.079,-96.053,-43.574,178.844,5.948,149.407
C08485=1152.084,-96.302,-43.565,178.842,5.948,149.408
C08486=1152.090,-96.553,-43.555,178.839,5.947,149.408
C08487=1152.095,-96.802,-43.546,178.837,5.947,149.409
C08488=1152.100,-97.052,-43.537,178.835,5.947,149.409
C08489=1152.105,-97.301,-43.527,178.833,5.946,149.410
C08490=1152.111,-97.551,-43.518,178.831,5.946,149.411
C08491=1152.117,-97.801,-43.508,178.829,5.945,149.411
C08492=1152.121,-98.051,-43.499,178.827,5.945,149.412
C08493=1152.127,-98.300,-43.490,178.825,5.945,149.412
C08494=1152.132,-98.551,-43.480,178.822,5.944,149.413
C08495=1152.138,-98.800,-43.471,178.821,5.944,149.413
C08496=1152.142,-99.050,-43.462,178.818,5.944,149.414
C08497=1152.148,-99.300,-43.452,178.816,5.943,149.414
C08498=1152.154,-99.550,-43.443,178.814,5.943,149.415
C08499=1152.158,-99.799,-43.434,178.812,5.942,149.415
C08500=1152.164,-100.049,-43.424,178.810,5.942,149.416
C08501=1152.169,-100.299,-43.415,178.808,5.942,149.416
C08502=1152.175,-100.549,-43.407,178.805,5.941,149.417
C08503=1152.180,-100.798,-43.396,178.804,5.941,149.418
C08504=1152.185,-101.048,-43.387,178.802,5.941,149.418
C08505=1152.191,-101.298,-43.379,178.800,5.941,149.419
C08506=1152.196,-101.548,-43.369,178.797,5.940,149.419
C08507=1152.201,-101.797,-43.359,178.795,5.940,149.420
C08508=1152.207,-102.047,-43.351,178.794,5.940,149.420
C08509=1152.212,-102.320,-43.341,178.791,5.939,149.421
C08510=1152.218,-102.591,-43.331,178.789,5.938,149.421
C08511=1152.225,-102.863,-43.320,178.787,5.939,149.422
C08512=1152.230,-103.136,-43.311,178.784,5.938,149.423
C08513=1152.235,-103.385,-43.301,178.782,5.937,149.423
C08514=1152.240,-103.635,-43.292,178.781,5.937,149.424
C08515=1152.246,-103.885,-43.283,178.778,5.937,149.424
C08516=1152.252,-104.135,-43.274,178.776,5.936,149.425
C08517=1152.257,-104.385,-43.265,178.774,5.936,149.425
C08518=1152.262,-104.635,-43.256,178.772,5.936,149.426
C08519=1152.267,-104.884,-43.247,178.770,5.936,149.426
C08520=1152.273,-105.134,-43.237,178.768,5.935,149.427
C08521=1152.278,-105.383,-43.229,178.765,5.934,149.427
C08522=1152.284,-105.633,-43.220,178.764,5.934,149.428
C08523=1152.289,-105.883,-43.211,178.761,5.934,149.429
C08524=1152.294,-106.133,-43.202,178.760,5.934,149.429
C08525=1152.300,-106.383,-43.192,178.757,5.933,149.430
C08526=1152.305,-106.633,-43.183,178.756,5.933,149.430
C08527=1152.310,-106.883,-43.175,178.754,5.933,149.431
C08528=1152.315,-107.132,-43.165,178.751,5.932,149.431
C08529=1152.320,-107.382,-43.156,178.749,5.932,149.432
C08530=1152.327,-107.631,-43.147,178.747,5.932,149.432
C08531=1152.332,-107.881,-43.138,178.746,5.932,149.433
C08532=1152.337,-108.131,-43.129,178.743,5.931,149.433
C08533=1152.342,-108.381,-43.120,178.741,5.931,149.434
C08534=1152.347,-108.630,-43.111,178.739,5.931,149.434
C08535=1152.352,-108.880,-43.102,178.737,5.930,149.435
C08536=1152.358,-109.131,-43.093,178.735,5.930,149.435
C08537=1152.364,-109.380,-43.084,178.733,5.929,149.436
C08538=1152.369,-109.629,-43.075,178.731,5.929,149.437
C08539=1152.375,-109.879,-43.067,178.729,5.929,149.437
C08540=1152.380,-110.129,-43.058,178.727,5.928,149.438
C08541=1152.385,-110.379,-43.049,178.725,5.928,149.438
C08542=1152.390,-110.629,-43.040,178.722,5.928,149.439
C08543=1152.396,-110.879,-43.030,178.721,5.928,149.439
C08544=1152.402,-111.128,-43.022,178.719,5.927,149.440
C08545=1152.407,-111.378,-43.013,178.717,5.927,149.440
C08546=1152.412,-111.628,-43.004,178.715,5.926,149.441
C08547=1152.417,-111.878,-42.995,178.713,5.927,149.441
C08548=1152.422,-112.128,-42.986,178.710,5.926,149.442
C08549=1152.428,-112.377,-42.977,178.708,5.925,149.442
C08550=1152.433,-112.627,-42.969,178.707,5.925,149.443
C08551=1152.438,-112.876,-42.960,178.705,5.924,149.443
C08552=1152.444,-113.126,-42.951,178.702,5.925,149.444
C08553=1152.450,-113.377,-42.942,178.700,5.924,149.445
C08554=1152.455,-113.627,-42.933,178.699,5.924,149.445
C08555=1152.461,-113.876,-42.925,178.696,5.923,149.446
C08556=1152.466,-114.126,-42.916,178.695,5.923,149.446
C08557=1152.471,-114.376,-42.907,178.693,5.923,149.447
C08558=1152.476,-114.626,-42.898,178.690,5.922,149.447
C08559=1152.481,-114.876,-42.889,178.688,5.922,149.448
C08560=1152.487,-115.125,-42.881,178.686,5.922,149.448
C08561=1152.492,-115.375,-42.872,178.685,5.922,149.449
C08562=1152.498,-115.625,-42.864,178.682,5.921,149.449
C08563=1152.503,-115.875,-42.855,178.680,5.921,149.450
C08564=1152.509,-116.124,-42.846,178.678,5.921,149.450
C08565=1152.514,-116.374,-42.837,178.677,5.921,149.451
C08566=1152.519,-116.624,-42.828,178.674,5.920,149.451
C08567=1152.524,-116.874,-42.820,178.673,5.920,149.452
C08568=1152.530,-117.123,-42.811,178.671,5.919,149.452
C08569=1152.535,-117.373,-42.803,178.668,5.919,149.453
C08570=1152.541,-117.623,-42.794,178.666,5.919,149.454
C08571=1152.546,-117.873,-42.785,178.664,5.918,149.454
C08572=1152.552,-118.122,-42.776,178.662,5.918,149.455
C08573=1152.557,-118.372,-42.768,178.660,5.917,149.455
C08574=1152.562,-118.622,-42.759,178.659,5.917,149.455
C08575=1152.567,-118.872,-42.750,178.656,5.917,149.456
C08576=1152.573,-119.121,-42.742,178.654,5.917,149.457
C08577=1152.578,-119.371,-42.733,178.652,5.916,149.457
C08578=1152.584,-119.622,-42.725,178.651,5.916,149.458
C08579=1152.589,-119.872,-42.716,178.648,5.916,149.458
C08580=1152.595,-120.121,-42.707,178.647,5.916,149.459
C08581=1152.600,-120.371,-42.699,178.645,5.915,149.459
C08582=1152.605,-120.621,-42.690,178.643,5.915,149.460
C08583=1152.611,-120.870,-42.682,178.640,5.914,149.460
C08584=1152.616,-121.120,-42.673,178.639,5.915,149.461
C08585=1152.621,-121.370,-42.664,178.637,5.914,149.461
C08586=1152.626,-121.620,-42.656,178.634,5.913,149.462
C08587=1152.632,-121.869,-42.648,178.633,5.913,149.462
C08588=1152.637,-122.119,-42.639,178.631,5.912,149.463
C08589=1152.643,-122.369,-42.631,178.628,5.913,149.463
C08590=1152.648,-122.619,-42.622,178.626,5.912,149.464
C08591=1152.654,-122.868,-42.613,178.625,5.912,149.464
C08592=1152.659,-123.118,-42.605,178.622,5.911,149.465
C08593=1152.665,-123.368,-42.597,178.621,5.911,149.465
C08594=1152.670,-123.618,-42.588,178.619,5.911,149.466
C08595=1152.675,-123.868,-42.579,178.617,5.911,149.466
C08596=1152.680,-124.117,-42.572,178.614,5.910,149.467
C08597=1152.686,-124.367,-42.563,178.613,5.910,149.468
C08598=1152.691,-124.618,-42.555,178.611,5.910,149.468
C08599=1152.697,-124.867,-42.546,178.609,5.910,149.469
C08600=1152.702,-125.117,-42.537,178.607,5.909,149.469
C08601=1152.708,-125.367,-42.529,178.605,5.909,149.470
C08602=1152.713,-125.616,-42.520,178.603,5.908,149.470
C08603=1152.718,-125.866,-42.512,178.601,5.908,149.471
C08604=1152.723,-126.116,-42.504,178.599,5.908,149.471
C08605=1152.729,-126.365,-42.495,178.597,5.908,149.472
C08606=1152.734,-126.616,-42.487,178.595,5.907,149.472
C08607=1152.740,-126.866,-42.478,178.593,5.907,149.473
C08608=1152.745,-127.115,-42.470,178.591,5.906,149.473
C08609=1152.750,-127.365,-42.462,178.590,5.906,149.474
C08610=1152.755,-127.615,-42.453,178.587,5.906,149.474
C08611=1152.761,-127.865,-42.446,178.586,5.906,149.475
C08612=1152.766,-128.114,-42.437,178.584,5.905,149.475
C08613=1152.346,-128.125,-42.479,178.580,5.909,149.477
C08614=1152.340,-127.876,-42.488,178.582,5.909,149.476
C08615=1152.335,-127.626,-42.496,178.584,5.910,149.476
C08616=1152.329,-127.376,-42.505,178.586,5.910,149.476
C08617=1152.324,-127.126,-42.512,178.588,5.910,149.475
C08618=1152.319,-126.876,-42.521,178.589,5.910,149.475
C08619=1152.313,-126.627,-42.529,178.592,5.911,149.474
C08620=1152.308,-126.377,-42.538,178.594,5.911,149.473
C08621=1152.303,-126.127,-42.547,178.596,5.911,149.473
C08622=1152.297,-125.878,-42.554,178.598,5.911,149.472
C08623=1152.292,-125.628,-42.563,178.600,5.912,149.472
C08624=1152.287,-125.377,-42.571,178.601,5.912,149.471
C08625=1152.281,-125.128,-42.580,178.604,5.913,149.471
C08626=1152.276,-124.878,-42.589,178.605,5.913,149.470
C08627=1152.270,-124.628,-42.597,178.607,5.914,149.470
C08628=1152.264,-124.379,-42.605,178.609,5.914,149.469
C08629=1152.260,-124.129,-42.614,178.612,5.914,149.469
C08630=1152.254,-123.879,-42.622,178.613,5.914,149.468
C08631=1152.249,-123.629,-42.630,178.615,5.915,149.468
C08632=1152.244,-123.380,-42.639,178.617,5.915,149.467
C08633=1152.238,-123.129,-42.647,178.619,5.915,149.467
C08634=1152.232,-122.880,-42.656,178.621,5.915,149.466
C08635=1152.227,-122.630,-42.665,178.623,5.916,149.466
C08636=1152.222,-122.380,-42.673,178.625,5.916,149.465
C08637=1152.216,-122.130,-42.681,178.627,5.916,149.465
C08638=1152.211,-121.881,-42.690,178.629,5.916,149.464
C08639=1152.206,-121.630,-42.698,178.631,5.917,149.464
C08640=1152.200,-121.381,-42.706,178.633,5.917,149.463
C08641=1152.195,-121.131,-42.715,178.635,5.918,149.463
C08642=1152.190,-120.882,-42.724,178.636,5.918,149.462
C08643=1152.184,-120.631,-42.732,178.639,5.919,149.462
C08644=1152.179,-120.382,-42.741,178.641,5.918,149.461
C08645=1152.173,-120.132,-42.750,178.643,5.919,149.460
C08646=1152.168,-119.882,-42.758,178.645,5.920,149.460
C08647=1152.162,-119.633,-42.767,178.647,5.920,149.459
C08648=1152.157,-119.383,-42.776,178.649,5.920,149.459
C08649=1152.152,-119.133,-42.784,178.651,5.920,149.459
C08650=1152.147,-118.883,-42.793,178.653,5.921,149.458
C08651=1152.141,-118.633,-42.801,178.655,5.921,149.457
C08652=1152.136,-118.383,-42.810,178.657,5.921,149.457
C08653=1152.130,-118.134,-42.819,178.659,5.921,149.456
C08654=1152.125,-117.884,-42.828,178.661,5.922,149.456
C08655=1152.119,-117.635,-42.836,178.662,5.922,149.455
C08656=1152.114,-117.384,-42.845,178.665,5.923,149.455
C08657=1152.109,-117.134,-42.853,178.667,5.922,149.454
C08658=1152.104,-116.884,-42.862,178.669,5.923,149.454
C08659=1152.098,-116.635,-42.871,178.670,5.923,149.453
C08660=1152.093,-116.385,-42.880,178.673,5.924,149.453
C08661=1152.087,-116.135,-42.888,178.675,5.925,149.452
C08662=1152.082,-115.885,-42.897,178.676,5.925,149.452
C08663=1152.076,-115.636,-42.905,178.679,5.925,149.451
C08664=1152.071,-115.386,-42.914,178.681,5.925,149.451
C08665=1152.066,-115.136,-42.923,178.683,5.926,149.450
C08666=1152.061,-114.886,-42.932,178.685,5.926,149.450
C08667=1152.056,-114.636,-42.941,178.687,5.926,149.449
C08668=1152.050,-114.387,-42.949,178.689,5.926,149.448
C08669=1152.044,-114.137,-42.958,178.691,5.927,149.448
C08670=1152.039,-113.887,-42.967,178.693,5.927,149.447
C08671=1152.034,-113.637,-42.975,178.695,5.927,149.447
C08672=1152.028,-113.388,-42.984,178.697,5.928,149.446
C08673=1152.023,-113.138,-42.993,178.699,5.928,149.446
C08674=1152.018,-112.888,-43.002,178.701,5.928,149.445
C08675=1152.012,-112.638,-43.011,178.703,5.928,149.445
C08676=1152.007,-112.388,-43.020,178.705,5.929,149.444
C08677=1152.002,-112.138,-43.029,178.707,5.929,149.444
C08678=1151.996,-111.889,-43.038,178.709,5.930,149.443
C08679=1151.991,-111.639,-43.047,178.712,5.930,149.443
C08680=1151.986,-111.390,-43.055,178.713,5.930,149.442
C08681=1151.980,-111.140,-43.064,178.715,5.931,149.442
C08682=1151.975,-110.890,-43.073,178.717,5.931,149.441
C08683=1151.969,-110.641,-43.082,178.719,5.932,149.441
C08684=1151.964,-110.391,-43.091,178.721,5.931,149.440
C08685=1151.958,-110.141,-43.100,178.723,5.932,149.439
C08686=1151.953,-109.891,-43.109,178.725,5.932,149.439
C08687=1151.948,-109.641,-43.118,178.727,5.933,149.438
C08688=1151.943,-109.391,-43.127,178.729,5.933,149.438
C08689=1151.938,-109.141,-43.136,178.731,5.933,149.437
C08690=1151.932,-108.892,-43.144,178.734,5.934,149.437
C08691=1151.926,-108.642,-43.154,178.735,5.934,149.436
C08692=1151.921,-108.392,-43.163,178.737,5.935,149.436
C08693=1151.916,-108.142,-43.172,178.739,5.935,149.435
C08694=1151.911,-107.892,-43.180,178.742,5.935,149.435
C08695=1151.905,-107.643,-43.189,178.744,5.936,149.434
C08696=1151.900,-107.393,-43.198,178.745,5.936,149.434
C08697=1151.894,-107.143,-43.208,178.748,5.936,149.433
C08698=1151.889,-106.893,-43.216,178.749,5.936,149.433
C08699=1151.883,-106.644,-43.225,178.752,5.937,149.432
C08700=1151.878,-106.394,-43.234,178.754,5.937,149.431
C08701=1151.873,-106.144,-43.243,178.756,5.937,149.431
C08702=1151.867,-105.894,-43.252,178.758,5.938,149.430
C08703=1151.862,-105.644,-43.262,178.760,5.938,149.430
C08704=1151.857,-105.395,-43.271,178.762,5.938,149.429
C08705=1151.852,-105.145,-43.280,178.764,5.938,149.429
C08706=1151.847,-104.895,-43.289,178.766,5.939,149.428
C08707=1151.841,-104.645,-43.298,178.768,5.940,149.428
C08708=1151.835,-104.396,-43.307,178.770,5.940,149.427
C08709=1151.830,-104.146,-43.316,178.772,5.940,149.427
C08710=1151.825,-103.897,-43.325,178.774,5.940,149.426
C08711=1151.819,-103.646,-43.335,178.776,5.941,149.426
C08712=1151.814,-103.397,-43.344,178.779,5.941,149.425
C08713=1151.809,-103.147,-43.353,178.781,5.941,149.424
C08714=1151.803,-102.875,-43.363,178.783,5.942,149.424
C08715=1151.798,-102.602,-43.372,178.785,5.942,149.423
C08716=1151.792,-102.330,-43.383,178.787,5.942,149.423
C08717=1151.785,-102.059,-43.393,178.790,5.943,149.422
C08718=1151.780,-101.809,-43.402,178.792,5.944,149.422
C08719=1151.775,-101.559,-43.411,178.793,5.944,149.421
C08720=1151.770,-101.309,-43.420,178.796,5.944,149.421
C08721=1151.764,-101.060,-43.430,178.798,5.945,149.420
C08722=1151.759,-100.810,-43.439,178.800,5.945,149.419
C08723=1151.754,-100.560,-43.448,178.802,5.945,149.419
C08724=1151.748,-100.310,-43.457,178.804,5.945,149.418
C08725=1151.743,-100.061,-43.467,178.806,5.946,149.418
C08726=1151.738,-99.811,-43.476,178.809,5.946,149.417
C08727=1151.732,-99.561,-43.485,178.810,5.946,149.417
C08728=1151.727,-99.311,-43.494,178.812,5.947,149.416
C08729=1151.722,-99.061,-43.504,178.815,5.948,149.416
C08730=1151.716,-98.811,-43.513,178.817,5.948,149.415
C08731=1151.711,-98.561,-43.522,178.819,5.948,149.415
C08732=1151.706,-98.312,-43.531,178.820,5.948,149.414
C08733=1151.700,-98.062,-43.541,178.823,5.949,149.414
C08734=1151.695,-97.812,-43.550,178.825,5.949,149.413
C08735=1151.689,-97.562,-43.560,178.827,5.949,149.412
C08736=1151.684,-97.313,-43.569,178.829,5.950,149.412
C08737=1151.679,-97.063,-43.578,178.832,5.951,149.411
C08738=1151.673,-96.813,-43.588,178.833,5.950,149.411
C08739=1151.668,-96.564,-43.597,178.836,5.951,149.410
C08740=1151.663,-96.314,-43.606,178.837,5.951,149.410
C08741=1151.658,-96.064,-43.616,178.840,5.952,149.409
C08742=1151.652,-95.814,-43.625,178.842,5.952,149.409
C08743=1151.646,-95.564,-43.635,178.844,5.952,149.408
C08744=1151.642,-95.315,-43.644,178.846,5.953,149.408
C08745=1151.636,-95.065,-43.653,178.849,5.953,149.407
C08746=1151.631,-94.815,-43.663,178.850,5.953,149.406
C08747=1151.626,-94.566,-43.672,178.852,5.954,149.406
C08748=1151.620,-94.315,-43.682,178.854,5.954,149.405
C08749=1151.615,-94.066,-43.691,178.857,5.955,149.405
C08750=1151.609,-93.816,-43.701,178.859,5.955,149.404
C08751=1151.604,-93.567,-43.711,178.860,5.955,149.404
C08752=1151.598,-93.317,-43.720,178.863,5.956,149.403
C08753=1151.594,-93.066,-43.729,178.865,5.956,149.403
C08754=1151.589,-92.817,-43.739,178.867,5.956,149.402
C08755=1151.583,-92.567,-43.748,178.869,5.957,149.402
C08756=1151.578,-92.318,-43.758,178.872,5.958,149.401
C08757=1151.572,-92.067,-43.768,178.873,5.957,149.400
C08758=1151.567,-91.818,-43.777,178.875,5.958,149.400
C08759=1151.561,-91.568,-43.787,178.878,5.959,149.399
C08760=1151.556,-91.319,-43.796,178.880,5.959,149.399
C08761=1151.551,-91.069,-43.806,178.882,5.959,149.398
C08762=1151.546,-90.819,-43.815,178.884,5.960,149.398
C08763=1151.540,-90.569,-43.825,178.886,5.960,149.397
C08764=1151.535,-90.320,-43.834,178.888,5.960,149.397
C08765=1151.530,-90.069,-43.844,178.891,5.961,149.396
C08766=1151.525,-89.820,-43.854,178.893,5.961,149.395
C08767=1151.519,-89.570,-43.863,178.895,5.962,149.395
C08768=1151.514,-89.320,-43.873,178.896,5.962,149.394
C08769=1151.508,-89.070,-43.883,178.899,5.962,149.394
C08770=1151.503,-88.821,-43.892,178.901,5.963,149.393
C08771=1151.498,-88.572,-43.902,178.903,5.963,149.393
C08772=1151.492,-88.321,-43.912,178.905,5.963,149.392
C08773=1151.488,-88.071,-43.922,178.908,5.964,149.391
C08774=1151.482,-87.821,-43.931,178.909,5.964,149.391
C08775=1151.477,-87.572,-43.941,178.912,5.965,149.391
C08776=1151.471,-87.322,-43.950,178.914,5.965,149.390
C08777=1151.466,-87.073,-43.960,178.916,5.965,149.389
C08778=1151.460,-86.823,-43.970,178.918,5.966,149.389
C08779=1151.455,-86.573,-43.979,178.920,5.966,149.388
C08780=1151.450,-86.323,-43.990,178.923,5.967,149.388
C08781=1151.445,-86.073,-44.000,178.924,5.967,149.387
C08782=1151.439,-85.824,-44.009,178.927,5.968,149.387
C08783=1151.434,-85.574,-44.019,178.929,5.968,149.386
C08784=1151.429,-85.325,-44.029,178.931,5.968,149.385
C08785=1151.423,-85.075,-44.038,178.933,5.969,149.385
C08786=1151.418,-84.824,-44.049,178.936,5.969,149.384
C08787=1151.413,-84.575,-44.058,178.937,5.969,149.384
C08788=1151.407,-84.325,-44.068,178.940,5.970,149.383
C08789=1151.402,-84.076,-44.077,178.942,5.970,149.383
C08790=1151.397,-83.826,-44.088,178.944,5.970,149.382
C08791=1151.392,-83.575,-44.098,178.946,5.971,149.382
C08792=1151.387,-83.326,-44.107,178.948,5.972,149.381
C08793=1151.381,-83.077,-44.117,178.950,5.971,149.380
C08794=1151.375,-82.826,-44.127,178.953,5.972,149.380
C08795=1151.370,-82.577,-44.136,178.955,5.973,149.379
C08796=1151.365,-82.327,-44.147,178.957,5.972,149.379
C08797=1151.360,-82.077,-44.157,178.959,5.973,149.378
C08798=1151.355,-81.828,-44.166,178.961,5.974,149.378
C08799=1151.349,-81.578,-44.176,178.964,5.974,149.377
C08800=1151.343,-81.328,-44.187,178.965,5.974,149.377
C08801=1151.339,-81.079,-44.197,178.968,5.975,149.376
C08802=1151.334,-80.829,-44.207,178.970,5.975,149.375
C08803=1151.328,-80.579,-44.216,178.972,5.975,149.375
C08804=1151.322,-80.329,-44.226,178.974,5.976,149.374
C08805=1151.318,-80.079,-44.236,178.977,5.977,149.374
C08806=1151.312,-79.830,-44.247,178.978,5.977,149.373
C08807=1151.307,-79.580,-44.257,178.981,5.977,149.373
C08808=1151.301,-79.330,-44.266,178.983,5.978,149.372
C08809=1151.296,-79.080,-44.276,178.985,5.978,149.372
C08810=1151.291,-78.831,-44.286,178.987,5.978,149.371
C08811=1151.285,-78.581,-44.297,178.990,5.979,149.370
C08812=1151.280,-78.332,-44.306,178.992,5.980,149.370
C08813=1151.275,-78.082,-44.317,178.993,5.980,149.369
C08814=1151.269,-77.831,-44.326,178.996,5.980,149.369
C08815=1151.264,-77.582,-44.337,178.998,5.981,149.368
C08816=1151.259,-77.333,-44.346,179.001,5.982,149.368
C08817=1151.254,-77.082,-44.357,179.003,5.981,149.367
C08818=1151.247,-76.812,-44.368,179.005,5.982,149.367
C08819=1151.242,-76.540,-44.379,179.007,5.982,149.366
C08820=1151.236,-76.269,-44.390,179.010,5.983,149.365
C08821=1151.230,-75.997,-44.400,179.012,5.983,149.365
C08822=1151.225,-75.747,-44.411,179.015,5.984,149.364
C08823=1151.220,-75.498,-44.421,179.017,5.984,149.363
C08824=1151.214,-75.248,-44.431,179.019,5.985,149.363
C08825=1151.209,-74.999,-44.441,179.021,5.985,149.363
C08826=1151.204,-74.749,-44.451,179.023,5.985,149.362
C08827=1151.199,-74.499,-44.462,179.025,5.986,149.361
C08828=1151.193,-74.250,-44.472,179.027,5.986,149.361
C08829=1151.188,-73.999,-44.482,179.030,5.987,149.360
C08830=1151.182,-73.750,-44.493,179.032,5.987,149.360
C08831=1151.178,-73.501,-44.502,179.034,5.988,149.359
C08832=1151.173,-73.250,-44.513,179.037,5.988,149.358
C08833=1151.167,-73.001,-44.523,179.039,5.989,149.358
C08834=1151.161,-72.751,-44.533,179.040,5.989,149.358
C08835=1151.156,-72.501,-44.544,179.043,5.989,149.357
C08836=1151.151,-72.251,-44.554,179.045,5.990,149.356
C08837=1151.145,-72.002,-44.564,179.047,5.991,149.356
C08838=1151.140,-71.752,-44.575,179.049,5.990,149.355
C08839=1151.135,-71.502,-44.584,179.052,5.991,149.355
C08840=1151.130,-71.253,-44.595,179.054,5.991,149.354
C08841=1151.125,-71.003,-44.605,179.057,5.992,149.353
C08842=1151.119,-70.753,-44.615,179.058,5.992,149.353
C08843=1151.114,-70.503,-44.626,179.061,5.993,149.352
C08844=1151.109,-70.253,-44.636,179.063,5.993,149.352
C08845=1151.103,-70.004,-44.646,179.065,5.994,149.351
C08846=1151.098,-69.753,-44.657,179.067,5.994,149.351
C08847=1151.093,-69.505,-44.668,179.069,5.994,149.350
C08848=1151.087,-69.255,-44.678,179.072,5.995,149.350
C08849=1151.082,-69.005,-44.689,179.074,5.996,149.349
C08850=1151.076,-68.755,-44.699,179.076,5.996,149.348
C08851=1151.071,-68.505,-44.710,179.078,5.996,149.348
C08852=1151.066,-68.255,-44.720,179.081,5.997,149.347
C08853=1151.061,-68.006,-44.729,179.083,5.998,149.347
C08854=1151.056,-67.756,-44.740,179.085,5.997,149.346
C08855=1151.051,-67.507,-44.751,179.087,5.998,149.346
C08856=1151.046,-67.257,-44.761,179.089,5.999,149.345
C08857=1151.040,-67.007,-44.772,179.092,5.999,149.344
C08858=1151.034,-66.758,-44.782,179.094,6.000,149.344
C08859=1151.029,-66.507,-44.792,179.096,6.000,149.343
C08860=1151.024,-66.259,-44.803,179.099,6.000,149.343
C08861=1151.019,-66.008,-44.814,179.101,6.001,149.342
C08862=1151.014,-65.759,-44.824,179.103,6.001,149.342
C08863=1151.009,-65.508,-44.835,179.105,6.001,149.341
C08864=1151.003,-65.259,-44.845,179.107,6.002,149.341
C08865=1150.998,-65.009,-44.856,179.110,6.003,149.340
C08866=1150.993,-64.760,-44.866,179.112,6.003,149.339
C08867=1150.987,-64.510,-44.877,179.114,6.004,149.339
C08868=1150.982,-64.260,-44.887,179.116,6.004,149.338
C08869=1150.976,-64.011,-44.899,179.118,6.004,149.338
C08870=1150.971,-63.761,-44.909,179.121,6.005,149.337
C08871=1150.965,-63.511,-44.919,179.123,6.006,149.337
C08872=1150.960,-63.261,-44.930,179.125,6.006,149.336
C08873=1150.955,-63.012,-44.941,179.128,6.006,149.335
C08874=1150.950,-62.762,-44.952,179.130,6.007,149.335
C08875=1150.945,-62.512,-44.962,179.132,6.007,149.334
C08876=1150.940,-62.262,-44.973,179.135,6.008,149.334
C08877=1150.934,-62.013,-44.983,179.136,6.008,149.333
C08878=1150.929,-61.763,-44.994,179.139,6.008,149.333
C08879=1150.924,-61.514,-45.005,179.141,6.009,149.332
C08880=1150.919,-61.263,-45.015,179.143,6.010,149.332
C08881=1150.913,-61.014,-45.026,179.146,6.010,149.331
C08882=1150.909,-60.764,-45.037,179.148,6.010,149.330
C08883=1150.902,-60.514,-45.048,179.150,6.011,149.330
C08884=1150.897,-60.264,-45.058,179.152,6.011,149.329
C08885=1150.892,-60.015,-45.069,179.155,6.012,149.329
C08886=1150.887,-59.765,-45.080,179.157,6.013,149.328
C08887=1150.882,-59.515,-45.090,179.159,6.013,149.328
C08888=1150.877,-59.266,-45.101,179.162,6.013,149.327
C08889=1150.871,-59.016,-45.111,179.164,6.014,149.326
C08890=1150.867,-58.767,-45.123,179.166,6.015,149.326
C08891=1150.860,-58.517,-45.133,179.169,6.015,149.325
C08892=1150.856,-58.267,-45.145,179.170,6.015,149.325
C08893=1150.851,-58.017,-45.155,179.173,6.015,149.324
C08894=1150.845,-57.767,-45.166,179.175,6.016,149.324
C08895=1150.840,-57.518,-45.177,179.177,6.017,149.323
C08896=1150.835,-57.268,-45.187,179.180,6.017,149.322
C08897=1150.829,-57.018,-45.199,179.182,6.018,149.322
C08898=1150.824,-56.769,-45.209,179.184,6.018,149.321
C08899=1150.819,-56.519,-45.220,179.186,6.018,149.321
C08900=1150.814,-56.269,-45.231,179.189,6.019,149.320
C08901=1150.809,-56.020,-45.242,179.191,6.020,149.319
C08902=1150.803,-55.769,-45.253,179.193,6.020,149.319
C08903=1150.798,-55.520,-45.264,179.196,6.021,149.318
C08904=1150.793,-55.270,-45.275,179.198,6.021,149.318
C08905=1150.788,-55.021,-45.286,179.200,6.022,149.317
C08906=1150.782,-54.771,-45.296,179.202,6.022,149.317
C08907=1150.777,-54.521,-45.308,179.205,6.023,149.316
C08908=1150.771,-54.272,-45.318,179.207,6.023,149.315
C08909=1150.767,-54.022,-45.330,179.210,6.024,149.315
C08910=1150.762,-53.772,-45.341,179.211,6.024,149.314
C08911=1150.756,-53.522,-45.352,179.214,6.024,149.314
C08912=1150.751,-53.273,-45.363,179.216,6.025,149.313
C08913=1150.745,-53.023,-45.373,179.219,6.026,149.313
C08914=1150.741,-52.774,-45.384,179.221,6.026,149.312
C08915=1150.735,-52.523,-45.396,179.223,6.027,149.312
C08916=1150.730,-52.274,-45.406,179.225,6.027,149.311
C08917=1150.725,-52.025,-45.418,179.227,6.027,149.310
C08918=1150.719,-51.774,-45.429,179.230,6.028,149.310
C08919=1150.714,-51.525,-45.440,179.232,6.029,149.309
C08920=1150.709,-51.275,-45.451,179.234,6.029,149.309
C08921=1150.703,-51.026,-45.462,179.237,6.030,149.308
C08922=1150.698,-50.755,-45.474,179.239,6.031,149.308
C08923=1150.692,-50.484,-45.486,179.242,6.031,149.307
C08924=1150.686,-50.214,-45.498,179.245,6.031,149.306
C08925=1150.680,-49.943,-45.510,179.247,6.032,149.306
C08926=1150.676,-49.693,-45.521,179.249,6.033,149.305
C08927=1150.670,-49.444,-45.533,179.251,6.033,149.305
C08928=1150.665,-49.194,-45.544,179.254,6.033,149.304
C08929=1150.660,-48.944,-45.555,179.256,6.034,149.303
C08930=1150.654,-48.695,-45.566,179.258,6.035,149.303
C08931=1150.649,-48.445,-45.577,179.261,6.035,149.302
C08932=1150.644,-48.195,-45.588,179.263,6.036,149.302
C08933=1150.638,-47.946,-45.600,179.266,6.036,149.301
C08934=1150.634,-47.696,-45.611,179.268,6.037,149.301
C08935=1150.628,-47.446,-45.623,179.270,6.037,149.300
C08936=1150.623,-47.197,-45.633,179.272,6.037,149.299
C08937=1150.618,-46.947,-45.644,179.274,6.038,149.299
C08938=1150.612,-46.697,-45.656,179.277,6.039,149.298
C08939=1150.608,-46.447,-45.667,179.279,6.039,149.298
C08940=1150.601,-46.197,-45.678,179.282,6.040,149.297
C08941=1150.597,-45.948,-45.690,179.284,6.040,149.297
C08942=1150.591,-45.698,-45.701,179.286,6.041,149.296
C08943=1150.587,-45.448,-45.713,179.288,6.041,149.295
C08944=1150.581,-45.199,-45.724,179.290,6.042,149.295
C08945=1150.576,-44.949,-45.736,179.293,6.042,149.294
C08946=1150.571,-44.699,-45.746,179.295,6.043,149.294
C08947=1150.565,-44.450,-45.758,179.298,6.043,149.293
C08948=1150.560,-44.200,-45.769,179.300,6.044,149.293
C08949=1150.555,-43.950,-45.781,179.302,6.045,149.292
C08950=1150.550,-43.701,-45.792,179.305,6.045,149.291
C08951=1150.544,-43.452,-45.804,179.307,6.046,149.291
C08952=1150.539,-43.202,-45.815,179.309,6.046,149.290
C08953=1150.534,-42.951,-45.826,179.311,6.046,149.290
C08954=1150.529,-42.702,-45.837,179.314,6.047,149.289
C08955=1150.523,-42.452,-45.849,179.316,6.048,149.289
C08956=1150.518,-42.203,-45.860,179.318,6.048,149.288
C08957=1150.513,-41.953,-45.872,179.321,6.049,149.287
C08958=1150.508,-41.703,-45.883,179.323,6.050,149.287
C08959=1150.503,-41.453,-45.895,179.326,6.050,149.286
C08960=1150.497,-41.204,-45.906,179.328,6.051,149.286
C08961=1150.492,-40.954,-45.918,179.331,6.051,149.285
C08962=1150.487,-40.705,-45.929,179.333,6.052,149.284
C08963=1150.482,-40.455,-45.941,179.334,6.052,149.284
C08964=1150.477,-40.205,-45.952,179.337,6.052,149.283
C08965=1150.471,-39.956,-45.964,179.339,6.053,149.283
C08966=1150.466,-39.706,-45.976,179.342,6.054,149.282
C08967=1150.461,-39.457,-45.987,179.344,6.054,149.282
C08968=1150.456,-39.207,-45.999,179.347,6.055,149.281
C08969=1150.451,-38.957,-46.010,179.349,6.056,149.280
C08970=1150.445,-38.707,-46.022,179.351,6.056,149.280
C08971=1150.440,-38.458,-46.033,179.354,6.057,149.279
C08972=1150.435,-38.208,-46.045,179.356,6.058,149.279
C08973=1150.429,-37.958,-46.057,179.359,6.058,149.278
C08974=1150.425,-37.709,-46.068,179.361,6.059,149.278
C08975=1150.419,-37.459,-46.080,179.363,6.058,149.277
C08976=1150.414,-37.209,-46.092,179.365,6.059,149.277
C08977=1150.408,-36.960,-46.103,179.368,6.060,149.276
C08978=1150.403,-36.710,-46.115,179.370,6.060,149.275
C08979=1150.398,-36.460,-46.126,179.372,6.061,149.275
C08980=1150.393,-36.210,-46.138,179.375,6.062,149.274
C08981=1150.387,-35.960,-46.150,179.377,6.062,149.274
C08982=1150.383,-35.711,-46.161,179.380,6.063,149.273
C08983=1150.378,-35.461,-46.174,179.382,6.064,149.272
C08984=1150.372,-35.211,-46.186,179.385,6.064,149.272
C08985=1150.367,-34.963,-46.197,179.387,6.065,149.271
C08986=1150.361,-34.713,-46.208,179.389,6.065,149.271
C08987=1150.356,-34.463,-46.220,179.392,6.066,149.270
C08988=1150.351,-34.213,-46.232,179.394,6.067,149.270
C08989=1150.346,-33.963,-46.244,179.396,6.067,149.269
C08990=1150.341,-33.714,-46.256,179.399,6.068,149.269
C08991=1150.335,-33.464,-46.268,179.401,6.068,149.268
C08992=1150.331,-33.214,-46.279,179.403,6.068,149.267
C08993=1150.325,-32.964,-46.291,179.406,6.069,149.267
C08994=1150.320,-32.714,-46.303,179.408,6.070,149.266
C08995=1150.315,-32.466,-46.315,179.410,6.070,149.265
C08996=1150.309,-32.216,-46.327,179.413,6.071,149.265
C08997=1150.304,-31.966,-46.338,179.415,6.072,149.265
C08998=1150.299,-31.716,-46.350,179.417,6.072,149.264
C08999=1150.294,-31.467,-46.362,179.420,6.073,149.263
C09000=1150.289,-31.217,-46.374,179.422,6.073,149.263
C09001=1150.283,-30.967,-46.386,179.424,6.074,149.262
C09002=1150.278,-30.717,-46.398,179.427,6.074,149.261
C09003=1150.273,-30.468,-46.410,179.429,6.075,149.261
C09004=1150.268,-30.218,-46.422,179.432,6.076,149.260
C09005=1150.263,-29.969,-46.434,179.434,6.076,149.260
C09006=1150.257,-29.719,-46.446,179.436,6.077,149.259
C09007=1150.252,-29.469,-46.458,179.439,6.078,149.259
C09008=1150.247,-29.220,-46.470,179.441,6.078,149.258
C09009=1150.242,-28.970,-46.481,179.444,6.079,149.257
C09010=1150.237,-28.720,-46.494,179.446,6.080,149.257
C09011=1150.231,-28.470,-46.506,179.449,6.080,149.256
C09012=1150.226,-28.221,-46.518,179.451,6.081,149.256
C09013=1150.222,-27.972,-46.530,179.454,6.081,149.255
C09014=1150.216,-27.722,-46.542,179.456,6.082,149.255
C09015=1150.211,-27.472,-46.554,179.458,6.083,149.254
C09016=1150.206,-27.222,-46.566,179.461,6.083,149.254
C09017=1150.200,-26.972,-46.578,179.463,6.084,149.253
C09018=1150.195,-26.723,-46.591,179.465,6.085,149.252
C09019=1150.190,-26.473,-46.602,179.468,6.085,149.252
C09020=1150.185,-26.224,-46.615,179.470,6.086,149.251
C09021=1150.180,-25.974,-46.626,179.472,6.087,149.251
C09022=1150.174,-25.724,-46.638,179.475,6.087,149.250
C09023=1150.169,-25.475,-46.651,179.477,6.088,149.250
C09024=1150.164,-25.225,-46.663,179.480,6.088,149.249
C09025=1150.159,-24.976,-46.675,179.482,6.089,149.248
C09026=1150.153,-24.705,-46.688,179.485,6.089,149.248
C09027=1150.147,-24.436,-46.701,179.487,6.090,149.247
C09028=1150.142,-24.166,-46.715,179.490,6.091,149.246
C09029=1150.136,-23.895,-46.728,179.492,6.091,149.246
C09030=1150.131,-23.645,-46.740,179.494,6.092,149.245
C09031=1150.127,-23.396,-46.752,179.497,6.092,149.245
C09032=1150.121,-23.146,-46.764,179.499,6.093,149.244
C09033=1150.116,-22.897,-46.777,179.501,6.094,149.244
C09034=1150.111,-22.648,-46.789,179.504,6.094,149.243
C09035=1150.105,-22.398,-46.801,179.506,6.095,149.243
C09036=1150.100,-22.149,-46.814,179.509,6.095,149.242
C09037=1150.095,-21.899,-46.826,179.511,6.096,149.241
C09038=1150.090,-21.649,-46.838,179.514,6.097,149.241
C09039=1150.084,-21.399,-46.850,179.516,6.098,149.240
C09040=1150.079,-21.150,-46.863,179.519,6.099,149.239
C09041=1150.074,-20.900,-46.875,179.521,6.100,149.239
C09042=1150.069,-20.651,-46.887,179.524,6.100,149.238
C09043=1150.064,-20.401,-46.900,179.526,6.101,149.238
C09044=1150.059,-20.151,-46.912,179.528,6.102,149.237
C09045=1150.054,-19.902,-46.925,179.531,6.102,149.237
C09046=1150.048,-19.652,-46.936,179.533,6.103,149.236
C09047=1150.043,-19.402,-46.949,179.536,6.103,149.236
C09048=1150.038,-19.153,-46.962,179.538,6.104,149.235
C09049=1150.033,-18.903,-46.974,179.541,6.104,149.234
C09050=1150.027,-18.654,-46.986,179.543,6.105,149.234
C09051=1150.023,-18.404,-46.999,179.546,6.106,149.233
C09052=1150.017,-18.154,-47.011,179.548,6.106,149.233
C09053=1150.012,-17.904,-47.024,179.550,6.107,149.232
C09054=1150.006,-17.655,-47.037,179.553,6.108,149.232
C09055=1150.001,-17.405,-47.049,179.555,6.108,149.231
C09056=1149.996,-17.156,-47.061,179.558,6.109,149.230
C09057=1149.991,-16.906,-47.074,179.560,6.110,149.230
C09058=1149.986,-16.656,-47.087,179.562,6.110,149.229
C09059=1149.981,-16.406,-47.099,179.565,6.111,149.229
C09060=1149.976,-16.157,-47.111,179.567,6.111,149.228
C09061=1149.971,-15.908,-47.124,179.569,6.112,149.228
C09062=1149.965,-15.658,-47.137,179.572,6.113,149.227
C09063=1149.961,-15.408,-47.149,179.574,6.113,149.226
C09064=1149.955,-15.158,-47.162,179.577,6.114,149.226
C09065=1149.950,-14.909,-47.175,179.580,6.115,149.225
C09066=1149.945,-14.659,-47.187,179.582,6.116,149.225
C09067=1149.939,-14.409,-47.199,179.584,6.117,149.224
C09068=1149.935,-14.159,-47.212,179.587,6.117,149.224
C09069=1149.929,-13.910,-47.225,179.589,6.118,149.223
C09070=1149.924,-13.661,-47.237,179.592,6.119,149.222
C09071=1149.918,-13.411,-47.250,179.594,6.119,149.222
C09072=1149.913,-13.162,-47.263,179.596,6.120,149.221
C09073=1149.909,-12.911,-47.275,179.599,6.120,149.221
C09074=1149.903,-12.662,-47.288,179.601,6.121,149.220
C09075=1149.898,-12.413,-47.301,179.604,6.122,149.219
C09076=1149.893,-12.163,-47.313,179.606,6.122,149.219
C09077=1149.888,-11.913,-47.327,179.609,6.123,149.218
C09078=1149.883,-11.664,-47.339,179.611,6.124,149.218
C09079=1149.878,-11.414,-47.352,179.614,6.125,149.217
C09080=1149.873,-11.165,-47.364,179.616,6.126,149.217
C09081=1149.868,-10.914,-47.377,179.618,6.126,149.216
C09082=1149.862,-10.665,-47.390,179.621,6.127,149.216
C09083=1149.857,-10.415,-47.403,179.623,6.128,149.215
C09084=1149.852,-10.166,-47.415,179.626,6.128,149.214
C09085=1149.847,-9.916,-47.428,179.628,6.129,149.214
C09086=1149.841,-9.666,-47.441,179.631,6.129,149.213
C09087=1149.836,-9.417,-47.454,179.633,6.130,149.213
C09088=1149.832,-9.167,-47.467,179.636,6.131,149.212
C09089=1149.826,-8.918,-47.479,179.638,6.131,149.212
C09090=1149.821,-8.668,-47.493,179.640,6.132,149.211
C09091=1149.815,-8.419,-47.505,179.643,6.133,149.210
C09092=1149.811,-8.169,-47.518,179.646,6.134,149.210
C09093=1149.805,-7.919,-47.531,179.648,6.135,149.209
C09094=1149.800,-7.670,-47.544,179.650,6.136,149.209
C09095=1149.795,-7.420,-47.557,179.653,6.136,149.208
C09096=1149.790,-7.171,-47.570,179.655,6.137,149.208
C09097=1149.784,-6.921,-47.583,179.658,6.137,149.207
C09098=1149.780,-6.671,-47.596,179.660,6.138,149.206
C09099=1149.775,-6.422,-47.608,179.663,6.138,149.206
C09100=1149.769,-6.172,-47.622,179.665,6.140,149.205
C09101=1149.765,-5.923,-47.635,179.668,6.140,149.205
C09102=1149.760,-5.673,-47.648,179.670,6.141,149.204
C09103=1149.754,-5.424,-47.661,179.673,6.142,149.203
C09104=1149.749,-5.174,-47.674,179.675,6.143,149.203
C09105=1149.743,-4.924,-47.687,179.678,6.143,149.202
C09106=1149.738,-4.675,-47.700,179.680,6.144,149.202
C09107=1149.734,-4.425,-47.713,179.682,6.145,149.201
C09108=1149.728,-4.175,-47.726,179.685,6.145,149.201
C09109=1149.723,-3.926,-47.739,179.687,6.147,149.200
C09110=1149.718,-3.676,-47.752,179.690,6.147,149.200
C09111=1149.713,-3.427,-47.765,179.692,6.148,149.199
C09112=1149.708,-3.177,-47.778,179.695,6.148,149.198
C09113=1149.702,-2.927,-47.792,179.697,6.149,149.198
C09114=1149.697,-2.678,-47.804,179.700,6.150,149.197
C09115=1149.693,-2.428,-47.818,179.702,6.150,149.197
C09116=1149.687,-2.179,-47.831,179.705,6.152,149.196
C09117=1149.682,-1.929,-47.844,179.707,6.152,149.196
C09118=1149.677,-1.679,-47.857,179.710,6.153,149.195
C09119=1149.672,-1.430,-47.870,179.712,6.154,149.194
C09120=1149.667,-1.180,-47.884,179.715,6.154,149.194
C09121=1149.661,-0.931,-47.897,179.717,6.155,149.193
C09122=1149.656,-0.680,-47.910,179.719,6.156,149.193
C09123=1149.651,-0.431,-47.923,179.722,6.157,149.192
C09124=1149.645,-0.182,-47.937,179.725,6.158,149.192
C09125=1149.641,0.068,-47.950,179.727,6.158,149.191
C09126=1149.635,0.318,-47.963,179.729,6.159,149.191
C09127=1149.631,0.567,-47.977,179.732,6.159,149.190
C09128=1149.625,0.817,-47.990,179.734,6.160,149.189
C09129=1149.620,1.067,-48.003,179.737,6.161,149.189
C09130=1149.614,1.335,-48.017,179.740,6.162,149.188
C09131=1149.609,1.605,-48.031,179.742,6.163,149.188
C09132=1149.604,1.875,-48.046,179.745,6.163,149.187
C09133=1149.598,2.144,-48.060,179.748,6.165,149.186
C09134=1149.593,2.393,-48.074,179.750,6.165,149.186
C09135=1149.588,2.643,-48.087,179.753,6.166,149.185
C09136=1149.582,2.893,-48.100,179.755,6.166,149.185
C09137=1149.578,3.142,-48.114,179.757,6.167,149.184
C09138=1149.572,3.392,-48.127,179.761,6.169,149.183
C09139=1149.567,3.641,-48.141,179.763,6.169,149.183
C09140=1149.562,3.891,-48.154,179.766,6.170,149.182
C09141=1149.557,4.141,-48.167,179.768,6.171,149.182
C09142=1149.552,4.390,-48.181,179.770,6.171,149.181
C09143=1149.546,4.640,-48.194,179.773,6.172,149.181
C09144=1149.542,4.889,-48.208,179.775,6.173,149.180
C09145=1149.536,5.139,-48.221,179.778,6.174,149.179
C09146=1149.532,5.388,-48.235,179.780,6.175,149.179
C09147=1149.526,5.638,-48.248,179.783,6.175,149.178
C09148=1149.521,5.888,-48.262,179.785,6.176,149.178
C09149=1149.517,6.138,-48.275,179.788,6.177,149.177
C09150=1149.511,6.387,-48.289,179.790,6.178,149.177
C09151=1149.506,6.637,-48.303,179.793,6.179,149.176
C09152=1149.501,6.886,-48.316,179.795,6.179,149.176
C09153=1149.496,7.136,-48.330,179.797,6.180,149.175
C09154=1149.491,7.385,-48.343,179.801,6.181,149.174
C09155=1149.486,7.635,-48.356,179.803,6.182,149.174
